(* CODESYS project TerminalApp.project
   Title: Терминал моечного поста
   Version: 0.0.0.1
   Company: ООО АСУ

Project tree, tasks and I/O mapping:
  CompWin : CODESYS Control for Raspberry Pi SL, 3S - Smart Software Solutions GmbH, version 3.5.11.60
    application AppTerminalPost
      libraries: Standard, * (System); Serial Communication, 3.5.7.0 (3S - Smart Software Solutions GmbH); Memory, 3.5.7.0 (3S - Smart Software Solutions GmbH); VisuDialogs, * (System); Time and Date, 3.5.7.0 (3S - Smart Software Solutions GmbH); BASIC, 3.3.3.0 (OSCAT); Standard64, * (System); Util, * (System); SysCom, 3.5.5.0 (System); SysProcess, 3.5.7.0 (System); SysTypes Interfaces, 3.5.2.0 (System); CmpChecksum, 3.5.5.0 (System); SysTime, 3.5.9.0 (System); CmpLog, 3.5.5.0 (System); Component Manager, * (System); CmpErrors Interfaces, * (System); CmpApp, 3.5.13.0 (System); File Access, 3.5.7.0 (3S - Smart Software Solutions GmbH); CmpCharDevice, 3.5.4.0 (3S - Smart Software Solutions GmbH)
      task MainTask (cyclic, interval 100 ms, priority 2) calls PLC_PRG, DeviceButtons, DeviceOut, SafePrg
      task TaskDevBanknote (cyclic, interval 4 ms, priority 1) calls DeviceBanknote [New Cash]
      task TaskDevCoin (cyclic, interval 5 ms, priority 4) calls DeviceCoin
      task TaskDevCard (cyclic, interval t#20ms, priority 3) calls DeviceCard
      task TaskDBG (cyclic, interval t#20ms, priority 1) calls DBG_PRG
      task NVLTask (cyclic, interval t#20ms, priority 1) calls DataToSpk, DataToUI, DataFromSpk
      task TaskPrinter (cyclic, interval t#20ms, priority 31) calls DevicePrinter
      program PLC_PRG [ST]: GetCurrentTime, SetValidComPorts, ControlCodesys
      Symbols
      data type EnumStatePost
      data type AppStatus
      Cash/
        program DeviceBanknote [ST]: GetCounterBanknote, IsCasetteDropped, IsBanknoteJammed, CollectCash, GetReceived
        data type CASHCODE_STATE
        data type CCNET_STATE
        function block COM_CONTROL [ST]: CLOSE, OPEN, SETTINGS
        data type _4BYTES_TO_REAL
        function _BUFFER_CLEAR [ST]
        data type _WORD_TO_2BYTES
        function block ANALYZE_DATA [ST]
        function BYTE_TO_STRH [ST]
        function block CashCode [ST]: CHECK_RESPONSE, GET_DATA_FROM_RESPONSE, GetCRC16, SET_ACK, SET_ENABLE_BILL_TYPES, SET_NSC, SET_PAKET, SET_POLL, SET_RESET, resetMoneyReceived, resetMoneyCnt
        data type COM_STATE
        data type DCON_STATE
        data type SET_4TM_STATE
        data type cacheCodeStatus
        data type CACHECODE_ERROR
        data type devBank
      DevCoin/
        program DeviceCoin [ST]: GetReceived, DbgInCoin, CollectCash, GetCounterCoin
        function block ccTalk [ST]: init, iterateAndUpdateStatus
        data type ccTalkStatus
        data type CCTALK_COIN_TYPES
        data type CCTALK_ERROR
        function block ccTalkSimpleCommand [ST]
        function block ccTalkReadBufferedCreditCommand [ST]
        data type ccTalkEvent
        function ccTalkCRC [ST]
        function ccTalkProcessReadBufferCreditTable [ST]
        function ccTalkGetNoDataCommandBuffer [ST]
      DevCard/
        function block Cards [ST]
        data type EnumCardType
        program DeviceCard [ST]: UnLockCard, DbgSetCard, GetTypeCard, TestValidComPort
        function block crt [ST]: init, iterateAndUpdateStatus, latchLock, latchRelease
        data type crtStatus
        data type CRT_CARD_STATE
        data type CRT_ERROR
        data type crtParametrizedCommand
        function block crtSimpleCommand [ST]
        function crtDecodeCardState [ST]
        function crtBCC [ST]
        function block crtInitCommand [ST]
      global variables GVL
      Debug/
        data type DebugStruct
        program DBG_PRG [ST]: GetInCoin, SetMode, GetInBanknote, UnLockCard
      DevButtons/
        program DeviceButtons [ST]: GetActiveButton
        data type EnumButton
      DevLamps/
        program DeviceLamps [ST]: SetLamps, SetAlarmLamps, SetIllumination, SetLampColor, SetLightTurbo
      Post/
        function block Post [ST]: ChangeMode, AddMoney, RemAmount, ResetModes, FormatModeFinInfo, StartWash, StopWash, SetCard, AvialableCardWork, InWaitModes, IsUnlocked, UnLock, IsReadyToWash, Init, EndCollectCash, BegCollectCash, EndFreemoney, BegFreemoney, InStopMode, OnFinButton, GeFundFromCollect, OnLowPower, SaveRetainVars, RestoreRetainVars, Shutdown, GetMessageInCash, GetMessageFunc, GetMessageCollect, GetFundTotal, GetRates, SaveNewRates, InPaidWashMode, InClearWashMode, GetMessageTotal, InServiceMode, SetSavedFund, SaveNewPause, GetPauseActiveClean, GetPauseFoam, GetPauseShampoo, SetLastInCash
        data type EnumMode
        function block EventMode [ST]: SetValues, ResetValues, StartMode, StopMode
        data type EnumLock
        program SafePrg [ST]
      Config/
        data type EnumInit
        function Initialisation [ST]
        function InitConfiguration [ST]
        function PostParamInit [ST]
        function PostStateInit [ST]
      DevOut/
        global variables NVL2UI
        program DeviceOut [ST]: SetOut
      global variables NVL_TO_SPK
      declarations NVL_FROM_SPK
      Traffic/
        program DataToSpk [ST]
        program DataFromSpk [ST]: GetConfirmedMode, GetAllowedButton, GetBonusValue, GetAllowedMode
        program DataToUI [ST]
      DevPrinter/
        data type PRINTER_FONT_CPI
        data type PRINTER_ERROR
        data type TEXT_ALIGNMENT
        data type PRINTER_FONT
        data type PRINTER_FONT_SIZE
        program DevicePrinter [ST]: printEncashment, PrintBill
        function block printReceipt [ST]
        function unicode2cp866 [ST]
        function unicodeSymbol2cp866 [ST]
        function block receiptBuffer [ST]: setFontCPI, setFontSize, clear, print, push_back, newline, push_back_array, setCP866Encoding, totalCut, initPrinter, ejectTicket, presentPageAndTimeoutRetract, setFontBold, setFontAlignment, println, printWithLeftPadding, print2Colsln, setFont, setFontSize2
      global variables SPK_DATA
      global variables PersistentVars
      program RetainManager [ST]
      function block StdLogger [ST]: AddLogEntry, debug, error, FB_Exit, FB_Init, info, warn
    SoftMotion General Axis Pool
    I²C
      I2C_master : I2C master, 3S - Smart Software Solutions GmbH, version 1.0.0.0
        UBRAIN1 : UBRAIN1, OOO ASU, version 1.1.0.0
            settings: I²C address = 5
    SPI
    GPIOs_A_B : GPIOs A/B, 3S - Smart Software Solutions GmbH, version 3.5.16.0
        unmapped channels: digital inputs (GPIO0..GPIO31), digital outputs (GPIO0..GPIO31)
    Onewire
    Camera device
      <Empty>
    Ethernet : Ethernet, 3S - Smart Software Solutions GmbH, version 3.5.16.0
        settings: IPAddress = [0,0,0,0]; SubnetMask = [0,0,0,0]; GatewayAddress = [0,0,0,0]; MACAddress = [16#00,16#00,16#00,16#00,16#00,16#00]; NetworkInterfaceName = 'eth0'; NetworkInterfaceName = "eth0"; SaveCommunicationSettings = FALSE
      ModbusTCP_Slave_Device : ModbusTCP Slave Device, 3S - Smart Software Solutions GmbH, version 3.5.16.0
          input  AppTerminalPost.SPK_DATA.gi_aAllowedFlags[0] : BOOL  // Регистры временного хранения.Регистры временного хранения.Bit0
          input  AppTerminalPost.SPK_DATA.gi_aAllowedFlags[1] : BOOL  // Регистры временного хранения.Регистры временного хранения.Bit1
          input  AppTerminalPost.SPK_DATA.gi_aAllowedFlags[2] : BOOL  // Регистры временного хранения.Регистры временного хранения.Bit2
          input  AppTerminalPost.SPK_DATA.gi_aAllowedFlags[3] : BOOL  // Регистры временного хранения.Регистры временного хранения.Bit3
          input  AppTerminalPost.SPK_DATA.gi_aAllowedFlags[4] : BOOL  // Регистры временного хранения.Регистры временного хранения.Bit4
          input  AppTerminalPost.SPK_DATA.gi_aAllowedFlags[5] : BOOL  // Регистры временного хранения.Регистры временного хранения.Bit5
          input  AppTerminalPost.SPK_DATA.gi_aAllowedFlags[6] : BOOL  // Регистры временного хранения.Регистры временного хранения.Bit6
          input  AppTerminalPost.SPK_DATA.gi_aAllowedFlags[7] : BOOL  // Регистры временного хранения.Регистры временного хранения.Bit7
          input  AppTerminalPost.SPK_DATA.gi_nCurFunction : WORD  // Регистры временного хранения.Регистры временного хранения
          output AppTerminalPost.SPK_DATA.go_postFunction : WORD  // Входные регистры.Входные регистры
          output AppTerminalPost.SPK_DATA.go_postCounterFund : WORD  // Входные регистры.Входные регистры
          unmapped channels: Регистры временного хранения, Входные регистры
  libraries: VisuSymbols, 3.5.10.0 (System)
  text list GlobalTextList
*)

// CompWin/AppTerminalPost/EnumStatePost
// Состояния поста
{attribute 'qualified_only'}
{attribute 'strict'}
TYPE EnumStatePost :
(
	IDLE	:= 0,	// Экран ожидания
	ADVERT	:= 100,	// Экран показа рекламы
	CARD	:= 200,	// Экран клиентской карты
	CASH	:= 300,	// Экран внесения денежных средств
	FUNC	:= 400,	// Экран функций
	FIN		:= 500,	// Экран окончания мойки
	CLEANUP	:= 600,	// Экран уборки
	ENCASH	:= 700,	// Экран инкассации
	STOP	:= 1000	// Экран состояния останова поста
);
END_TYPE

// CompWin/AppTerminalPost/Post/EnumMode
// Функции мойки
{attribute 'qualified_only'}
{attribute 'strict'}
TYPE EnumMode :
(
	FUNC		:= 0,	// терминал готов к включению функций
	
	ACTIVECLEAN	:= 1,	// Р1. ECO-power		2
	FOAM		:= 2,	// Р2. Пена				4
	SHAMPOO		:= 3,	// Р3. Шампунь			3
	COLDWATER	:= 4,	// Р4. Холодная вода	1
	HOTWATER	:= 5,	// Р5. Горячая вода		2
	WAX			:= 6,	// Р6. Воск				4
	OSMOSE		:= 7,	// Р7. Осмос			3
	PAUSE		:= 8,	// Пауза				4
	HIGHPRESSURE := 14, // ХВ высокого давления 
	
	IDLE		:= 9,	// терминал в ожидании клиентов
	ADVERT		:= 10,	// реклама	
	
	FIN			:= 500,	// Экран окончания мойки
	CLEANUP		:= 600,	// Экран уборки
	CASHCOLLECT	:= 700,	// Экран инкассации
	CASHCOLLECT_FIN	:= 710,	// Экран окончания инкассации
	FREEMONEY	:= 800,	// Экран добавления денег
	STOP		:= 1000	// Экран состояния останова поста

//	CARD	:= 200,	// Экран клиентской карты
//	CASH	:= 300,	// Экран внесения денежных средств
);
END_TYPE

// CompWin/AppTerminalPost/Config/EnumInit
// Кода возврата процедуры инициализации
{attribute 'qualified_only'}
{attribute 'strict'}
TYPE EnumInit :
(
	INIT_RET_FAIL       := 0, //      0 - инициализация закончилась с ошибкой
	INIT_RET_SUCC_RESET := 1, //      1 - инициализация успешно проведена, требуется перезапуск
	INIT_RET_SUCC       := 2, //      2 - инициализация успешно проведена, перезапуск не требуется
	INIT_RET_NO         := 3  //      3 - в инициализации не было необходимости
);
END_TYPE

// CompWin/AppTerminalPost/AppStatus
// Состояние приложения
TYPE AppStatus :
STRUCT
	startFlag: BOOL := TRUE;	// флаг начального запуска
	infoString: STRING := 'Starting ...';	// информация о состоянии приложения
	rebootFlag : BOOL := FALSE;	// флаг необходимости перезапуска
	
	errNimber: INT := 0;
	errString: STRING;
END_STRUCT
END_TYPE

// CompWin/AppTerminalPost/DevCard/EnumCardType
// Типы карт
{attribute 'qualified_only'}
{attribute 'strict'}
TYPE EnumCardType :
(
	UNDEFINED	:= 0,	// неопределённая карта (карта отсутствует)
	CLEANUP		:= 1,	// карта уборки
	CASHCOLLECT	:= 2,	// карта инкассации
	FREEMONEY	:= 3,	// карта добавления денег (бесплатной мойки)
	SERVICE		:= 4	// карта техслужбы
);
END_TYPE

// CompWin/AppTerminalPost/Cash/CASHCODE_STATE

TYPE CASHCODE_STATE :
(
	INIT,
	DISABLE,
	RESET,
	POLL,
	ENABLE_BILL_TYPES
);
END_TYPE

// CompWin/AppTerminalPost/Cash/CCNET_STATE

TYPE CCNET_STATE :
(
	INIT,
	IDLE,
	SEND_POLL,
	SEND_ENABLE_BILL_TYPES,
	SEND_COMMAND, //Command transmission
	SEND_ASC, //Подтверждаем получение
	SEND_NSC, //Не подтверждааем получение
	SEND_RESET, //reset
	RECEIVE_RESPONSE,
	RESPONSE_DELAY,
	WAIT_ENROLLMENT,
	WAIT_WRITE,
	POLLING_CYCLE_ENDS
	
	
);
END_TYPE

// CompWin/AppTerminalPost/DevCoin/ccTalkStatus
///element of ccTalk ReadBufferCredit (229) command output
TYPE ccTalkStatus :
STRUCT
	coinsReceived : ARRAY[0..5] OF BYTE;  //принятые монеты по номиналам
	coinsRejected : UINT;   //непринятые монеты
	moneyReceived : UINT;   //денег принято всего
	busy : BOOL := FALSE;  //cannot execute command
	error: CCTALK_ERROR;

	// количество монет в боксе
	countCoin: UINT := 0;
	// количества монет по номиналам
	receivedCoin1: UINT := 0;
	receivedCoin2: UINT := 0;
	receivedCoin5: UINT := 0;
	receivedCoin10: UINT := 0;
END_STRUCT
END_TYPE

// CompWin/AppTerminalPost/DevCoin/CCTALK_COIN_TYPES
TYPE CCTALK_COIN_TYPES :
(
//	COIN_1RUB := 16#1000 OR 16#0800,
//	COIN_2RUB := 16#4000 OR 16#2000,
//	COIN_5RUB := 16#0001 OR 16#8000,
//	COIN_10RUB := 16#0004 OR 16#0002

//	COIN_1RUB := 16#1000 OR 16#0800,
//	COIN_2RUB := 16#4000 OR 16#2000,
//	COIN_5RUB := 16#0001 OR 16#8000,
//	COIN_10RUB := 16#0001 OR 16#8000
	COIN_10RUB := 16#FFFF
	
) UINT;
END_TYPE

// CompWin/AppTerminalPost/DevCoin/CCTALK_ERROR
{attribute 'strict' := ''}
TYPE CCTALK_ERROR :
(
	CCTALK_NO_ERROR,
	CCTALK_OPEN_ERROR,
	CCTALK_INIT_PROC_NOT_CALLED
) BYTE;
END_TYPE

// CompWin/AppTerminalPost/DevCoin/ccTalkEvent
///element of ccTalk ReadBufferCredit (229) command output
TYPE ccTalkEvent :
STRUCT
	validationChannel: BYTE;
	errorCode: BYTE;
END_STRUCT
END_TYPE

// CompWin/AppTerminalPost/DevCard/crtStatus
///element of ccTalk ReadBufferCredit (229) command output
TYPE crtStatus :
STRUCT
	cardState: CRT_CARD_STATE := CRT_CARD_UNDEFINED;
	///cannot execute command
	busy: BOOL := FALSE;
	///is latch locked ?
	locked: BOOL := FALSE;
	error: CRT_ERROR;
	isInit : BOOL;
END_STRUCT
END_TYPE

// CompWin/AppTerminalPost/DevCard/CRT_CARD_STATE
{attribute 'strict' := ''}
TYPE CRT_CARD_STATE :
(
	CRT_CARD_UNDEFINED,
	CRT_CARD_INSIDE,
	CRT_RF_CARD_INSIDE,
	CRT_NO_CARD
);
END_TYPE

// CompWin/AppTerminalPost/DevCard/CRT_ERROR
{attribute 'strict' := ''}
TYPE CRT_ERROR :
(
	CRT_NO_ERROR,
	CRT_OPEN_ERROR,
	CRT_INIT_PROC_NOT_CALLED
);
END_TYPE

// CompWin/AppTerminalPost/DevCard/crtParametrizedCommand
///command and parameter for using in CRT protocol
TYPE crtParametrizedCommand :
STRUCT
	CM: BYTE;
	PM: BYTE;
END_STRUCT
END_TYPE

// CompWin/AppTerminalPost/Debug/DebugStruct
// Структура отладочной визуализации
TYPE DebugStruct :
STRUCT
//	Mode: EnumMode := EnumMode.WAIT;
	
	InBanknote: WORD := 0;
	
	InCoin: WORD := 0;
	
	CardType: EnumCardType := EnumCardType.UNDEFINED;
END_STRUCT
END_TYPE

// CompWin/AppTerminalPost/Cash/_4BYTES_TO_REAL
TYPE _4BYTES_TO_REAL :
UNION
	rValue :REAL;
	abyModbusReal : ARRAY [0..3] OF BYTE;
END_UNION
END_TYPE

// CompWin/AppTerminalPost/DevButtons/EnumButton
// функциональные кнопки
{attribute 'qualified_only'}
{attribute 'strict'}
TYPE EnumButton :
(
	NONE := 0,				// нет нажатой кнопки
	BTN_SHAMPOO := 1,		// Шампунь
	BTN_ACTIVECLEAN := 2,	// ECO-power
	BTN_FOAM := 3,			// Пена
	BTN_COLDWATER := 4,		// Холодная вода
	BTN_HOTWATER := 5,		// Горячая вода
	BTN_WAX := 6,			// Воск
	BTN_OSMOSE := 7,		// Осмос
	BTN_PAUSE := 8,			// Пауза
	BTN_PRINT := 9,			// Печать чека
	BTN_HIGHPRESSURE := 10	// Вызов оператора
);
END_TYPE

//VAR CONSTANT
//	BTN_FUNC_FIRST :BYTE := 1;
//	BTN_FUNC_LAST :BYTE := 8;
//	BTN_FIRST :BYTE := 1;
//	BTN_LAST :BYTE := 10;
//END_VAR

// CompWin/AppTerminalPost/Post/EnumLock
// замки поста
{attribute 'qualified_only'}
{attribute 'strict'}
TYPE EnumLock :
(
	LOCK_TOP := 1,	// 2#0100_0000,		// верхний замок
	LOCK_MID := 2	// 2#1000_0000		// средний замок
);
END_TYPE

// CompWin/AppTerminalPost/DevPrinter/PRINTER_FONT_CPI
{attribute 'strict' := ''}
TYPE PRINTER_FONT_CPI :
(
	CPI_SMALL := 0,
	CPI_BIG := 1,
	CPI_MEDIUM := 2
) BYTE;
END_TYPE

// CompWin/AppTerminalPost/DevPrinter/PRINTER_ERROR
{attribute 'strict' := ''}
TYPE PRINTER_ERROR :
(
	PRINTER_NO_ERROR,
	PRINTER_FILE_OPEN_ERROR,
	PRINTER_WRITE_ERROR
) BYTE;
END_TYPE

// CompWin/AppTerminalPost/DevPrinter/TEXT_ALIGNMENT
{attribute 'strict' := ''}
TYPE TEXT_ALIGNMENT :
(
	ALIGN_LEFT := 0,
	ALIGN_CENTER := 1,
	ALIGN_RIGHT := 2
) BYTE;
END_TYPE

// CompWin/AppTerminalPost/DevPrinter/PRINTER_FONT
{attribute 'strict' := ''}
TYPE PRINTER_FONT :
(
	FONT_A := 0,
	FONT_B := 1
) BYTE;
END_TYPE

// CompWin/AppTerminalPost/DevPrinter/PRINTER_FONT_SIZE
{attribute 'strict' := ''}
TYPE PRINTER_FONT_SIZE :
(
	FONT_SMALL := 1,
	FONT_BIG := 0
) BYTE;
END_TYPE

// CompWin/AppTerminalPost/Cash/_WORD_TO_2BYTES
TYPE _WORD_TO_2BYTES :
UNION
	wValue : WORD;
	abyWord : ARRAY [0..1] OF BYTE;
END_UNION
END_TYPE

// CompWin/AppTerminalPost/Cash/COM_STATE
TYPE COM_STATE :
(
	INITIALIZE := 00,
	WAITING_FOR_SIGNAL := 10,
	OPEN_PORT := 20,
	CLOSE_PORT := 30
);
END_TYPE

// CompWin/AppTerminalPost/Cash/DCON_STATE

TYPE DCON_STATE :
(
	CREATE_REQUEST := 00,
	SEND_REQUEST := 10,
	RECEIVE_RESPONSE := 20,
	RESPONSE_DELAY := 30,
	POLLING_CYCLE_ENDS := 40
);
END_TYPE

// CompWin/AppTerminalPost/Cash/SET_4TM_STATE
TYPE SET_4TM_STATE :
(
	CREATE_CHANNEL := 00,
	OPEN_CHANNEL := 10,
	RECEIVE_CHANNEL := 20,
	RESPONSE_DELAY_CHANNEL := 30,
	CREATE_REQUEST := 40,
	SEND_REQUEST := 50,
	RECEIVE_RESPONSE := 60,
	RESPONSE_DELAY := 70,
	POLLING_CYCLE_ENDS := 80
);
END_TYPE

// CompWin/AppTerminalPost/Cash/cacheCodeStatus
///element of ccTalk ReadBufferCredit (229) command output
TYPE cacheCodeStatus :
STRUCT
	///принятая купюра
	moneyReceived: UINT;
	///cannot execute command
	busy: BOOL := FALSE;
	error: CACHECODE_ERROR;
//	// количество купюр в боксе
//	countBanknote: UINT := 0;
	// состояние купюрника
	cashcodeStatus : WORD := 0;
	// ошибка купюрника
	cashcodeError : WORD := 0;

	// флаг снятия касетты
	casetteDropped : WORD := 0;
	// флаг зажёвывания банкноты
	banknoteJammed : WORD := 0;
	
	// количества купюр по номиналам
	receivedBanknote10: UINT := 0;
	receivedBanknote50: UINT := 0;
	receivedBanknote100: UINT := 0;
	receivedBanknote500: UINT := 0;
	receivedBanknote1000: UINT := 0;
	receivedBanknote5000: UINT := 0;
END_STRUCT
END_TYPE

// CompWin/AppTerminalPost/Cash/CACHECODE_ERROR
TYPE CACHECODE_ERROR :
(
	CACHECODE_NO_ERROR,
	CACHECODE_OPEN_ERROR
);
END_TYPE

// CompWin/AppTerminalPost/Cash/devBank
TYPE devBank :
(
	INIT := 0,
	CLOSE,
	OPEN,
	PROCESS
);
END_TYPE

// CompWin/AppTerminalPost/DevOut/NVL2UI
{attribute 'qualified_only'}
VAR_GLOBAL
	// номер поста
	postNumber: INT;
	
	// Состояние терминала: ожидание, функции, окончание мойки, уборка, инкассация, пополнение баланса оператором
	postMode: INT;
	// TYPE EnumMode :
	// (
	// 	FUNC		:= 0,	// терминал готов к включению функций
	// 	
	// 	ACTIVECLEAN	:= 1,	// Р1. ECO-power		2
	// 	FOAM		:= 2,	// Р2. Пена				4
	// 	SHAMPOO		:= 3,	// Р3. Шампунь			3
	// 	COLDWATER	:= 4,	// Р4. Холодная вода	1
	// 	HOTWATER	:= 5,	// Р5. Горячая вода		2
	// 	WAX			:= 6,	// Р6. Воск				4
	// 	OSMOSE		:= 7,	// Р7. Осмос			3
	// 	PAUSE		:= 8,	// Пауза				4
	// 	
	// 	IDLE		:= 9,	// терминал в ожидании клиентов
	// 	ADVERT		:= 10,	// реклама	
	// 	
	// 	FIN			:= 500,	// Экран окончания мойки
	// 	CLEANUP		:= 600,	// Экран уборки
	// 	CASHCOLLECT	:= 700,	// Экран инкассации
	// 	CASHCOLLECT_FIN	:= 710,	// Экран окончания инкассации
	// 	FREEMONEY	:= 800	// Экран добавления денег
	// 	STOP		:= 1000	// Экран состояния останова поста
	// );
	// END_TYPE

	// баланс
	postCounterFund: INT;

	// тип карты
	cardType: INT;
	// TYPE EnumCardType :
	// (
	// 	UNDEFINED	:= 0,	// неопределённая карта (карта отсутствует)
	// 	CLEANUP		:= 1,	// карта уборки
	// 	CASHCOLLECT	:= 2,	// карта инкассации
	// 	FREEMONEY	:= 3,	// карта добавления денег (бесплатной мойки)
	// 	SERVICE		:= 4	// карта техслужбы
	// );
	// END_TYPE	

	
	// нажатая кнопка
	buttonActive: INT;
	// TYPE EnumButton :
	// (
	// 	NONE := 0,				// нет нажатой кнопки
	// 	BTN_ACTIVECLEAN := 1,	// Р1. ECO-power
	// 	BTN_FOAM := 2,			// Р2. Пена
	// 	BTN_SHAMPOO := 3,		// Р3. Шампунь
	// 	BTN_COLDWATER := 4,		// Р4. Холодная вода
	// 	BTN_HOTWATER := 5,		// Р5. Горячая вода
	// 	BTN_WAX := 6,			// Р6. Воск
	// 	BTN_OSMOSE := 7,		// Р7. Осмос
	// 	BTN_PAUSE := 8,			// Пауза
	// 	BTN_PRINT := 9,			// Печать чека
	// 	BTN_HELP := 10			// Вызов оператора
	// );
	// END_TYPE
		
	// сумма внесения
	amountReceived: INT;
	
	
	// стоимость оконченной мойки
	costWash: INT;
	// сдача
	costChange: INT;
	// стоимость активной химии
	costActiveClean: INT;
	// стоимость пены
	costFoam: INT;
	// стоимость шампуня
	costShampoo: INT;
	// стоимость ХВ
	costColdWater: INT;
	// стоимость ГВ
	costHotWater: INT;
	// стоимость воска
	costWax: INT;
	// стоимость осмоса
	costOsmose: INT;
	// стоимость паузы
	costPause: INT;

	
	// состояние верхнего замка
	lockTop: INT;
	// состояние среднего замка
	lockMid: INT;
	// 1 - замок закрыт; 0 - замок открыт
END_VAR

// CompWin/AppTerminalPost/GVL
{attribute 'qualified_only'}
VAR_GLOBAL
	btn_1: BOOL;
	//cnt_1: INT;
	SetAlarmLamps: INT;
	
	printEncashmentReceipt : BOOL :=FALSE;
	
	glFlagStartVideo : ARRAY[0..10] OF BOOL;
	glFlagStartIdleVideo : BOOL;
	
END_VAR

// CompWin/AppTerminalPost/NVL_TO_SPK
{attribute 'qualified_only'}
VAR_GLOBAL
	// номер поста
	go_postNumber: INT;
	// выбранная функция
	go_postFunction: INT;
	// баланс поста
	go_postCounterFund: INT;
END_VAR

// CompWin/AppTerminalPost/NVL_FROM_SPK
//This gobal variable list is received via the network.
//Sender: Imported from file 'D:\lexadev\ЭкоМойки\gitrep\dev\TerminalController\NVL_Sender.gvl'
//Protocol: UDP

VAR_GLOBAL
	n_iCounter: INT;	
	n_aPostMode: ARRAY [0..5] OF INT;
	n_aAllowedFlags: ARRAY [0..5,1..7] OF BOOL;
END_VAR

// CompWin/AppTerminalPost/SPK_DATA
{attribute 'qualified_only'}
VAR_GLOBAL
	// to SPK
	go_postNumber: INT;
	go_postFunction: INT;
	go_postCounterFund: INT;
	go_counter: UINT;
	
	// from SPK
	gi_nCurFunction: INT;
	gi_aAllowedFlags: ARRAY [0..7] OF BOOL;

	// from AG
	// флаг необходимости применения тарифов от сервера
	// 1 - надо применить тарифы сервера, 0 - игнорировать
	gi_rateSave : WORD;
	
	// новые тарифы режимов от сервера 
	gi_rates : ARRAY [0 .. 8] OF WORD;
	
	// бонусы
	// текущий процент бонусов
	gi_bonusValue: WORD := 0;
	// час начала действия бонусов 24H
	gi_bonusStart: WORD := 22;
	// час окончания действия бонусов 24H
	gi_bonusStop: WORD := 6;
	
	
	// флаг необходимости применения пауз от сервера
	// 1 - надо применить паузы сервера, 0 - игнорировать
	gi_pauseSave : WORD;

	// паузы режимов в секундах
	gi_pauseActiveClean: WORD;
	gi_pauseFoam: WORD;
	gi_pauseShampoo: WORD;
	
	
	// to server
	counterBanknote10: WORD;
	counterBanknote50: WORD;
	counterBanknote100: WORD;
	counterBanknote500: WORD;
	counterBanknote1000: WORD;
	counterBanknote5000: WORD;

	counterCoin: WORD;
	counterCoin1: WORD;
	counterCoin2: WORD;
	counterCoin5: WORD;
	counterCoin10: WORD;
	
	// внесений с инкассации
	fundFromCollect: UINT;
	// внесений с начала работы
	fundTotal: UINT;

//	messageInCash: STRING;
//	messageFunc: STRING;
//	messageCollect: STRING;
	messageInCash: ARRAY[0..64] OF WORD;
	messageFunc:  ARRAY[0..64] OF WORD;
	messageCollect:  ARRAY[0..64] OF WORD;
	messageTotal:  ARRAY[0..64] OF WORD;
	
	// текущие тарифы
	currentRates : ARRAY[0..8] OF WORD;

	// ФЛАГИ КУПЮРНИКА
	// состояние купюрника
	cashcodeStatus : WORD := 0;
	// ошибка купюрника
	cashcodeError : WORD := 0;
	
	// флаг инкассации (отсоединения касетты)
	casetteDropped : WORD := 0;
	// флаг зажёвывания банкноты
	banknoteJammed : WORD := 0;
	
	// Флаги блокировки дверей
	lockTop : WORD := 1;
	lockMid : WORD := 1;
	
	// паузы режимов в секундах
	currentPauseActiveClean: WORD;
	currentPauseFoam: WORD;
	currentPauseShampoo: WORD;
END_VAR

// CompWin/AppTerminalPost/PersistentVars
{attribute 'qualified_only'}
VAR_GLOBAL PERSISTENT RETAIN
	// тотальная несбрасываемый счётчик выручки
	TotalFund : UINT := 0;	
	
	// total количества купюр по номиналам
	totalBanknote10: DWORD := 0;
	totalBanknote50: DWORD := 0;
	totalBanknote100: DWORD := 0;
	totalBanknote500: DWORD := 0;
	totalBanknote1k: DWORD := 0;
//	totalBanknote5000: DWORD := 0;

	// total количества монет по номиналам
//	totalCoin1: DWORD := 0;
//	totalCoin2: DWORD := 0;
//	totalCoin5: DWORD := 0;
	totalCoin10: DWORD := 0;

	//// выручка в посту (сбрасывается при инкассации)
	//CashFund : UINT := 0;
	
	// количества купюр по номиналам
	counterBanknote10: UINT := 0;
	counterBanknote50: UINT := 0;
	counterBanknote100: UINT := 0;
	counterBanknote500: UINT := 0;
	counterBanknote1000: UINT := 0;
//	counterBanknote5000: UINT := 0;

	// количества монет по номиналам
//	counterCoin1: UINT := 0;
//	counterCoin2: UINT := 0;
//	counterCoin5: UINT := 0;
	counterCoin10: UINT := 0;
	
	// количества купюр по номиналам до инкассации
	counterBefCollectBanknote10: UINT := 0;
	counterBefCollectBanknote50: UINT := 0;
	counterBefCollectBanknote100: UINT := 0;
	counterBefCollectBanknote500: UINT := 0;
	counterBefCollectBanknote1000: UINT := 0;
//	counterBefCollectBanknote5000: UINT := 0;

	// количества монет по номиналам до инкассации
//	counterBefCollectCoin1: UINT := 0;
//	counterBefCollectCoin2: UINT := 0;
//	counterBefCollectCoin5: UINT := 0;
	counterBefCollectCoin10: UINT := 0;
//	messageCollectCoin : STRING := '';
	
	// сообщение о внесении
	messageInCash: STRING[130] := '';
	// сообщение о функции
	messageFunc: STRING[130] := '';
	// сообщение об инкассации
	messageCollect: STRING[130] := '';
	// сообщение о тотальном счётчике
	messageTotal: STRING[130] := '';
	
	// тарифы функций 
	rates : ARRAY [0 .. 8] OF WORD := [
	2700, 	// ACTIVECLEAN	:= 1,	// Р1. ECO-power
	3300, 	// FOAM		:= ,	// Р2. Пена
	2300, 	// SHAMPOO		:= ,	// Р3. Вода + шампунь
	1500, 	// COLDWATER	:= 4,	// Р4. Холодная вода
	2400, 	// HOTWATER	:= 5,	// Р5. Горячая вода
	3600, 	// WAX			:= 6,	// Р6. Воск
	2700, 	// OSMOSE		:= 7,	// Р7. Осмос
	100,	// PAUSE		:= 8,	// пауза
	2100	// HIGHPRESSURE	:= 9,	// ХВ высокого давления
	];
	
	// сохранённый баланс  с меткой времени
	fundTime : DATE_AND_TIME;
	fundSaved100 : WORD;
	
	// адрес мойки
	washAddress : WSTRING := "Волгоград Жукова 55";
	// номер поста
	postNumber : INT := 0;
	
	// паузы режимов в секундах
	pauseActiveClean: TIME := T#10S;
	pauseFoam: TIME := T#0S;
	pauseShampoo: TIME := T#5S;
	flUseIdleVideo : BOOL := FALSE;
	
END_VAR

// CompWin/AppTerminalPost/PLC_PRG
PROGRAM PLC_PRG
VAR
	appStatus: AppStatus;	// состояние приложения
	
	post: Post;

	timStandbyTime: TIME := T#5S;	//Время в режиме ожидания (c)
	timAdvertisingTime: TIME := T#5S;	//Время в режиме рекламы (c)
	timFinTime: TIME := T#20S;	//Время в экране окончания мойки (c)
	
	timIdleFilterCash:		TIME;	//Фильтр задержки реакции на изменение сигналов внесения и уборки (с)
	timIdleFilterMode:		TIME;	//Фильтр задержки реакции на изменение сигналов режимов (с)
	
	receivedBanknote: WORD;
	receivedCoin: WORD;
	
   	getDT : DTU.GetDateAndTime;
	prevTime : DT;
	currentTime : DT;
	workSecond : DWORD;

	durationSecond: TIME;
	waitSecond: TIME;
	
	//amount : WORD;
	
	comPortCard : BYTE := 0;
	comPortCascode : BYTE := 0;
	
	ii : byte;
	InStopMode: INT;
	
	startTime : DT;
	
	// время начала режимов с задержкой
	startTm_ActiveClean: DT;
	startTm_Foam: DT;
	startTm_Shampoo: DT;
	fDelay: BOOL := FALSE;
	
	//Вспомогательные переменные
	udiResult: UDINT;
	udiTimeLocal : UDINT;
	timeDate: DATE_AND_TIME;
	
	bb : EnumButton;
	
	logger : StdLogger;
END_VAR

// в начале определить текущее время
currentTime := GetCurrentTime();
IF(currentTime > DT#1970-01-01-00:00:00)THEN
	// Начальная инициализация
	IF(appStatus.startFlag) THEN
		appStatus.infoString := Initialisation();
		
		RetainManager(ForceRestore := TRUE, ForceSave := FALSE);
	
		// Включить отладку
		//DBG_PRG.dbgProcess := TRUE;
		DBG_PRG.dbgProcess := FALSE;
		
		// инициализировать пост
		post.Init();
		
		// установить com порты
		SetValidComPorts();
		
		// восстановить сохранённый до перезапуска баланс
//		WHILE((currentTime = DT#1970-01-01-00:00:00) OR (idt < 1000))DO
//			currentTime := GetCurrentTime();
//			idt := idt + 1;
//		END_WHILE
		post.SetSavedFund(PersistentVars.fundTime, PersistentVars.fundSaved100 / 100.0);
	
		appStatus.startFlag := FALSE;
	END_IF
	
	//GVL.cnt_1 := GVL.cnt_1 + 1;
	
	currentTime := GetCurrentTime();
	IF(prevTime = DT#1970-01-01-00:00:00)THEN
		prevTime := currentTime;
	END_IF
	
	IF(startTime = DT#1970-01-01-00:00:00)THEN
		startTime := currentTime;
	END_IF
	
	// действия с периодичностью 1 секунда
	workSecond := TIME_TO_DWORD(currentTime - prevTime) / 1000;
	IF(workSecond > 0)THEN
		prevTime := currentTime;
		
		
	//	FOR ii := 1 TO 8 DO
	//		UBRAIN1.bColorButton[ii - 1] := DeviceLamps.COLOR_GREEN;
	//	END_FOR
	
	// учитывать задержку для определенных режимов	
	IF(NOT fDelay)THEN
		post.RemAmount(workSecond);
	END_IF
	
		// получить принятые купюры
		receivedBanknote := DeviceBanknote.GetReceived(); //xxx
		// получить принятые монеты
		receivedCoin := DeviceCoin.GetReceived();
	
		// увеличить сумму в посте
		//IF(receivedBanknote > 0 OR receivedCoin > 0)THEN
			post.AddMoney(receivedBanknote, receivedCoin);
		//END_IF
		
	//	IF(post.Mode <> DeviceButtons.Mode AND post.CounterFund > 0)THEN
	//		post.ChangeMode(DeviceButtons.Mode);
	//	END_IF
	
		// работа в режиме ожидания
		CASE post.Mode OF
	//		EnumMode.IDLE:
	//			waitSecond := timStandbyTime;
	//			durationSecond := currentTime - post.ModeStartTime;
	//			IF(durationSecond > waitSecond)THEN
	//				post.ChangeMode(EnumMode.ADVERT);
	//			END_IF;
	//		EnumMode.ADVERT:
	//			waitSecond := timAdvertisingTime;
	//			durationSecond := currentTime - post.ModeStartTime;
	//			IF(durationSecond > waitSecond)THEN
	//				post.ChangeMode(EnumMode.IDLE);
	//			END_IF;
			EnumMode.FIN:
				waitSecond := timFinTime;
				durationSecond := currentTime - post.ModeStartTime;
				IF(durationSecond > T#20S)THEN
					post.ChangeMode(EnumMode.IDLE);
				END_IF;
			EnumMode.CASHCOLLECT_FIN:
				waitSecond := timFinTime;
				durationSecond := currentTime - post.ModeStartTime;
				IF(durationSecond > T#5S)THEN
					post.ChangeMode(EnumMode.IDLE);
				END_IF;
		END_CASE
	END_IF
	
	// проверять CODESYS
	IF(post.InWaitModes())THEN
		ControlCodesys();
	END_IF
	
	// пост в останове
	IF(post.InStopMode())THEN
		// подсветка терминала
		DeviceLamps.SetIllumination(DeviceLamps.ILLUMINATION_COLOR_RED);
	END_IF
		
	// из режима ожидания переход к мойке
	IF(post.InWaitModes())THEN
		// подсветка терминала
		DeviceLamps.SetIllumination(DeviceLamps.ILLUMINATION_COLOR_LIGHTBLUE);
		GVL.glFlagStartIdleVideo := TRUE;	
		IF(post.IsReadyToWash()) THEN
			post.ChangeMode(EnumMode.FUNC);
		END_IF
	END_IF
	
	// работа в режиме мойки
	IF(post.IsReadyToWash())THEN
		// подсветка терминала
		IF(post.InClearWashMode())THEN
			// в режиме уборки - жёлтый
			DeviceLamps.SetIllumination(DeviceLamps.ILLUMINATION_COLOR_YELLOW);
		ELSE
			// основная подсветка в режиме мойки - зелёный
			DeviceLamps.SetIllumination(DeviceLamps.ILLUMINATION_COLOR_GREEN);
		END_IF
	
	//	CASE DeviceButtons.GetActiveButton() OF
		CASE DataFromSpk.GetConfirmedMode() OF
			EnumMode.ACTIVECLEAN:
				IF(startTm_ActiveClean = DT#1970-01-01-00:00:00)THEN
					startTm_ActiveClean := currentTime;
					fDelay := TRUE;
				ELSE
					durationSecond := currentTime - startTm_ActiveClean;
					IF(durationSecond >= post.GetPauseActiveClean())THEN
						fDelay := FALSE;
					END_IF;
				END_IF
				post.ChangeMode(EnumMode.ACTIVECLEAN);
			EnumMode.FOAM:
				IF(startTm_Foam = DT#1970-01-01-00:00:00)THEN
					startTm_Foam := currentTime;
					fDelay := TRUE;
				ELSE
					durationSecond := currentTime - startTm_Foam;
					IF(durationSecond >= post.GetPauseFoam())THEN
						fDelay := FALSE;
					END_IF;
				END_IF
				post.ChangeMode(EnumMode.FOAM);
			EnumMode.SHAMPOO:
				IF(startTm_Shampoo = DT#1970-01-01-00:00:00)THEN
					startTm_Shampoo := currentTime;
					fDelay := TRUE;
				ELSE
					durationSecond := currentTime - startTm_Shampoo;
					IF(durationSecond >= post.GetPauseShampoo())THEN
						fDelay := FALSE;
					END_IF;
				END_IF
				post.ChangeMode(EnumMode.SHAMPOO);
			EnumMode.COLDWATER:
				post.ChangeMode(EnumMode.COLDWATER);
			EnumMode.HOTWATER:
				post.ChangeMode(EnumMode.HOTWATER);
			EnumMode.WAX:
				post.ChangeMode(EnumMode.WAX);
			EnumMode.OSMOSE:
				post.ChangeMode(EnumMode.OSMOSE);
			EnumMode.PAUSE:
				post.ChangeMode(EnumMode.PAUSE);
			EnumMode.HIGHPRESSURE:
				post.ChangeMode(EnumMode.HIGHPRESSURE);
	//			IF(PLC_PRG.post.Mode = EnumMode.PAUSE)THEN
	//				post.ChangeMode(EnumMode.FIN);
	//			ELSE
	//				post.ChangeMode(EnumMode.PAUSE);
	//			END_IF
			10:
				// ошибка для выбранного режима
				DeviceLamps.SetAlarmLamps(DeviceButtons.GetActiveButton());
			11:
				// пост в останове
				DeviceLamps.SetAlarmLamps(0);
		END_CASE
		
		// сбросить время начала режимов с задержкой
		IF((DataFromSpk.GetConfirmedMode() <> EnumMode.ACTIVECLEAN) AND (DataFromSpk.GetConfirmedMode() <> EnumMode.FOAM) AND (DataFromSpk.GetConfirmedMode() <> EnumMode.SHAMPOO))THEN
			fDelay := FALSE;
		END_IF
		
		IF((startTm_ActiveClean <> DT#1970-01-01-00:00:00) AND (DataFromSpk.GetConfirmedMode() <> EnumMode.ACTIVECLEAN))THEN
			startTm_ActiveClean := DT#1970-01-01-00:00:00;
		END_IF

		IF((startTm_Foam <> DT#1970-01-01-00:00:00) AND (DataFromSpk.GetConfirmedMode() <> EnumMode.FOAM))THEN
			startTm_Foam := DT#1970-01-01-00:00:00;
		END_IF

		IF((startTm_Shampoo <> DT#1970-01-01-00:00:00) AND (DataFromSpk.GetConfirmedMode() <> EnumMode.SHAMPOO))THEN
			startTm_Shampoo := DT#1970-01-01-00:00:00;
		END_IF
	END_IF
	
	// сбросить время начала режимов с задержкой
	IF(NOT post.IsReadyToWash())THEN
		fDelay := FALSE;
		
		IF(startTm_ActiveClean <> DT#1970-01-01-00:00:00) THEN
			startTm_ActiveClean := DT#1970-01-01-00:00:00;
		END_IF

		IF(startTm_Foam <> DT#1970-01-01-00:00:00) THEN
			startTm_Foam := DT#1970-01-01-00:00:00;
		END_IF

		IF(startTm_Shampoo <> DT#1970-01-01-00:00:00) THEN
			startTm_Shampoo := DT#1970-01-01-00:00:00;
		END_IF
	END_IF
	
	// работа в режиме инкассации
	IF(post.Mode = EnumMode.CASHCOLLECT)THEN
		// из-за путаницы в кнопках в инкассации смотртеь на реально нажатую кнопку DeviceButtons.externalActiveButton 
		bb := DeviceButtons.externalActiveButton;
//		CASE DeviceButtons.GetActiveButton() OF
		CASE bb OF
			1:	//EnumButton.BTN_SHAMPOO:
				//// если пост закрыт, то открыть соответствующий замок
				//IF(NOT post.IsUnlocked(EnumLock.LOCK_TOP))THEN
					post.UnLock(EnumLock.LOCK_TOP, TRUE);
				//END_IF
			3:	//EnumButton.BTN_FOAM:
				//// если пост закрыт, то открыть соответствующий замок
				//IF(NOT post.IsUnlocked(EnumLock.LOCK_MID))THEN
					post.UnLock(EnumLock.LOCK_MID, TRUE);
				//END_IF
			2:	//EnumButton.BTN_ACTIVECLEAN:
				// инкассировать пост
				SysTimeRtcConvertUtcToLocal(SysTimeRtcGet(udiResult), udiTimeLocal);
				timeDate:= UDINT_TO_DT(udiTimeLocal);
		//sssxxx		//DevicePrinter.printEncashment(printingTime := OSCAT_BASIC.UTC_TO_LTIME(timeDate, DST_ENABLE :=0, TIME_ZONE_OFFSET:=DevicePrinter.TIME_ZONE_MINUTES_OFFSET), countBanknote10 := DeviceBanknote.GetCounterBanknote(10), countBanknote50 := DeviceBanknote.GetCounterBanknote(50), countBanknote100 := DeviceBanknote.GetCounterBanknote(100),  countCoin10 := DeviceCoin.GetCounterCoin(0));

				DeviceBanknote.CollectCash(); //xxx
				DeviceCoin.CollectCash();
		END_CASE
	END_IF
	
	// работа в режиме добавления денег (бесплатной мойки)
	IF(post.Mode = EnumMode.FREEMONEY)THEN
		CASE DeviceButtons.GetActiveButton() OF
			EnumButton.BTN_ACTIVECLEAN:
				// добавить 5 рублей
				post.AddMoney(5, 0);
			EnumButton.BTN_FOAM:
				// добавить 10 рублей
				post.AddMoney(10, 0);
			EnumButton.BTN_SHAMPOO:
				// добавить 50 рублей
				post.AddMoney(50, 0);
			EnumButton.BTN_COLDWATER:
				// добавить 100 рублей
				post.AddMoney(100, 0);
	//		EnumButton.BTN_PAUSE:
	//			post.EndFreemoney();
		END_CASE
	END_IF
END_IF

METHOD PUBLIC GetCurrentTime : DATE_AND_TIME
VAR
END_VAR
getDT.xExecute := NOT getDT.xDone;
getDT();
IF getDT.xError THEN
    ; // error handling
END_IF
IF getDT.xDone THEN
    // done without error
	currentTime := getDT.dtDateAndTime;
	 //eTZ := getdt.eTimezone;
END_IF

GetCurrentTime := currentTime;
END_METHOD

METHOD SetValidComPorts : BOOL
VAR_INPUT
END_VAR
VAR
	comPort : BYTE;
	portCard : BYTE := 0;
	portBanknote : BYTE := 0;
END_VAR

//DeviceBanknote.TestValidComPort(1);
//DeviceBanknote.TestValidComPort(2);
//DeviceBanknote.TestValidComPort(3);


//DeviceCard.TestValidComPort(10);
//DeviceCard.TestValidComPort(1);
//DeviceCard.TestValidComPort(2);
//DeviceCard.TestValidComPort(3);

//RETURN;

comPortCard := 2;
comPortCascode := 4;
RETURN;

(*
FOR comPort := 1 TO 10 DO
	IF(portCard = 0 AND comPort <> portBanknote)THEN
		IF(DeviceCard.TestValidComPort(comPort))THEN
			portCard := comPort;
		END_IF
	END_IF
	
	IF(portBanknote = 0 AND comPort <> portCard)THEN
		IF(DeviceBanknote.TestValidComPort(comPort))THEN
			portBanknote := comPort;
		END_IF
	END_IF
END_FOR

IF(portCard <> 0)THEN
	comPortCard := portCard;
END_IF

IF(portBanknote <> 0)THEN
	comPortCascode := portBanknote;
END_IF
*)
END_METHOD

METHOD ControlCodesys : BOOL
VAR

	ct : DATE_AND_TIME;

//    command:STRING:= 'sudo /etc/init.d/codesyscontrol restart; read -n1 -t1;';
//    command:STRING[256]:= 'sudo /etc/init.d/codesyscontrol stop && sudo /etc/init.d/codesyscontrol start && date';
    command:STRING[256]:= 'sudo /etc/init.d/codesyscontrol stop';
//    command:STRING:= 'touch /home/pi/mytest123.txt';
    res: SysCom.RTS_IEC_RESULT;
    outbuf:STRING(1000) := '';

END_VAR

ct := GetCurrentTime();
IF((ct - startTime) > T#60M AND NOT appStatus.rebootFlag) THEN
	appStatus.rebootFlag := TRUE;
	PersistentVars.fundSaved100 := 0;
	PersistentVars.fundTime := ct;
	// сохранить retain в файл
	post.SaveRetainVars();
	// выставить флаг необходимости считывания retain переменных из файла
	RetainManager.ForceRestore := TRUE;
	RetainManager.ForceSave := FALSE;
	appStatus.startFlag := TRUE;
	
//	SysProcess.SysProcessExecuteCommand(command, ADR(res));
	SysProcess.SysProcessExecuteCommand2(pszCommand:=command, pszStdOut:= outbuf, udiStdOutLen:= SIZEOF(outbuf), pResult:= ADR(res)); 
END_IF
END_METHOD

END_PROGRAM

// CompWin/AppTerminalPost/Config/Initialisation
// Основная функция инициализации приложения
FUNCTION Initialisation : STRING
VAR_INPUT
END_VAR
VAR
END_VAR

//// Главные установки
//InitBase();

// Инициализировать параметры и начальные значения поста
IF(InitConfiguration() < EnumInit.INIT_RET_SUCC) THEN
//    SDisplaySetError(0);
	Initialisation := 'Err InitConfiguration()';
    return;
END_IF

// Определить параметры поста
IF(PostParamInit() = 0)THEN
	Initialisation := 'Err PostParamInit()';
    RETURN;
END_IF;


//// Инициализировать прерывания таймера
//InitIRQTimer();
  
//// Инициализировать часы
//TimeInit();
  
// Определить состояние поста
PostStateInit();

Initialisation := 'Started';

END_FUNCTION

// CompWin/AppTerminalPost/Config/InitConfiguration
// Процедура инициализации устройства
FUNCTION InitConfiguration : EnumInit
VAR_INPUT
END_VAR
VAR
END_VAR

(*  // Проверить соответствие размеров буферов и структур
  if(SIZE_BUF_VER != sizeof(version_t))
    return INIT_RET_FAIL;
  
  if(SIZE_BUF_PARAM != sizeof(PostParam_t))
    return INIT_RET_FAIL;
  
  if(SIZE_BUF_STATE != sizeof(PostState_t))
    return INIT_RET_FAIL;

  if(SIZE_BUF_EVENT != sizeof(event_t))
    return INIT_RET_FAIL;
  

  // Проверить необходимость инициализации
  if(EEPROM_INIT_CODE == 0x00)
    return INIT_RET_NO;
  
  // Прописать версию ПО
  if(EEPROM_INIT_CODE & INIT_VER)
  {
    if(!MemIntWriteVersion(VERSION))
      return INIT_RET_FAIL;
  }
  
  // Прописать параметры поста
  if(EEPROM_INIT_CODE & INIT_PARAM)
  {
    if(!MemIntWritePostParam(pp))
      return INIT_RET_FAIL;
  }
  
  // Сбросить сохранённое состояние
  if(EEPROM_INIT_CODE & INIT_STATE)
  {
    if(!MemIntWritePostState(ps))
      return INIT_RET_FAIL;
  }
  
  // Сбросить кольцевой буфер, прописав ID следующего события и счётчики
  if(EEPROM_INIT_CODE & INIT_RB)
  {
    // если будет использована флэшка, то очищать её
    #ifdef MEM_FLASH
      MemFlashErase();
    #endif  // MEM_FLASH
      
    // Прописать инициализирующее событие
    uint32_t address = 0;
    #ifdef MEM_INT
      address = FADDR_INT_startRingBuffer;
    //#elif defined MEM_FLASH
    //  address = 0;
    #endif
    MemWriteEvent(address, e, 0);
    
    // Установить количество событий, сохранённых в кольцевом буфере, в 1
    MemIntWriteCountEvents(1);
  }
  
  // Сбросить состояние необходимости инициализации
  EEPROM_INIT_CODE = 0x00;
*)  
  InitConfiguration := EnumInit.INIT_RET_SUCC;

END_FUNCTION

// CompWin/AppTerminalPost/Config/PostParamInit
// Прочитать параметры поста
FUNCTION PostParamInit : BYTE
VAR_INPUT
END_VAR
VAR
END_VAR

  (*uint8_t pbuf[SIZE_BUF_PARAM];

  uint16_t address = FADDR_PARAM;
  
  for(int i = 0; i < sizeof(PostParam_t); i++)
  {
    pbuf[i] = FLASH_ReadByte(address + i);
  }
 
  memcpy(pparam, pbuf, sizeof(PostParam_t));
*)

PostParamInit := 1;

END_FUNCTION

// CompWin/AppTerminalPost/Config/PostStateInit
// Определить состояние поста
FUNCTION PostStateInit : BYTE
VAR_INPUT
END_VAR
VAR
END_VAR

(*
//  PostStateReset();
  
  PostStateRead();
  
  // При запуске всегда нет текущего режима (на флэшке сохранены только закончившиеся режимы)
  // Если не состояние уборки, то считаем, что платный режим
  PMResetCurrentMode(postState.stateKind != 2);
  
  event_t evnt;
  if(RBInitLastEventWithCounters(&evnt))
  {
    // Определить последнее внесение денег
    postState.counterBanknote = evnt.attrCash.counterBanknote;
    postState.counterCoin = evnt.attrCash.counterCoin;
  }

  switch(postState.stateKind)
  {
    case 1:
      // Продолжить сохранённое оставшееся оплаченое время
      if(postState.timerRemain > 0)
        PostTimerIncrement(postState.timerRemain);
      break;
    case 2:
      PMModeFreeSet(1);
      break;
    case 3:
      SDisplaySetCounter(postState.counterBanknote);
      break;
    case 4:
      SDisplaySetCounter(postState.counterCoin);
      break;
  }
*)

PostStateInit := 1;

END_FUNCTION

// CompWin/AppTerminalPost/RetainManager
PROGRAM RetainManager

VAR_INPUT
   RetainFilePathName : STRING := '/home/pi/ASU/AppTerminalPost.ret';
   SaveFilterTime : TIME := T#300MS;
   ForceSave : BOOL;
   ForceRestore : BOOL := TRUE;
   ForceBalance : BOOL := FALSE;
END_VAR
VAR
   pRetainFilePathName : POINTER TO STRING;
   pCurrentApp : POINTER TO APPLICATION;
   RetainAreaSize: __XWORD;
   pRetainArea: POINTER TO BYTE;
   dwCRCSave: DWORD;
   dwCRC: DWORD;
   TOF1 : TOF := (PT := SaveFilterTime);
   R_TRIG1: R_TRIG;
   AppGetCurrent: INT;
   
   
	synccmd: STRING := 'sync -f /home/pi/ASU/AppTerminalPost.ret';
	msg: WSTRING(255);
END_VAR
VAR_OUTPUT
   RTSIECResult : RTS_IEC_RESULT;   
   AttemptSaveCounter: INT;
   Init: BOOL := FALSE;
END_VAR

IF ForceRestore THEN
   pCurrentApp := CmpApp.AppGetCurrent(ADR(RTSIECResult));
   IF RTSIECResult<>0 THEN RETURN; END_IF
   RetainAreaSize := AppGetAreaSize(pApp:= pCurrentApp, uiType:= DA_RETAIN, pResult:= ADR(RTSIECResult));
   IF RTSIECResult<>0 THEN RETURN; END_IF
   pRetainArea := AppGetAreaAddress(pApp:= pCurrentApp, uiType:= DA_RETAIN, pResult:= ADR(RTSIECResult));
   IF RTSIECResult<>0 THEN RETURN; END_IF
   IF LEN(RetainFilePathName) <> 0 THEN
      pRetainFilePathName := ADR(RetainFilePathName);
   ELSE
      pRetainFilePathName := ADR(pCurrentApp^.szName);   
   END_IF
   RTSIECResult := AppRestoreRetainsFromFile(pCurrentApp, pRetainFilePathName^);   
	msg := "ForceRestore";
	PLC_PRG.logger.debug(msg);
   CASE RTSIECResult OF
      0: // #define ERR_OK 0x0000
			msg := "ForceRestore: ERR_OK";
			PLC_PRG.logger.debug(msg);
      16#1E: // #define ERR_SIGNATURE_MISMATCH 0x001E   /* Signature mismatch of an api function */
			msg := "ForceRestore: Signature mismatch of an api function";
			PLC_PRG.logger.debug(msg);
      16#32: // #define ERR_FILE_ERROR 0x0032   /* File error. e.g. cannot open a file for writing because it could be write protected */
			msg := "ForceRestore: File error. e.g. cannot open a file for writing because it could be write protected";
			PLC_PRG.logger.debug(msg);
   ELSE RETURN;
   END_CASE
   dwCRCSave := CRC32Finish(ulCRC:= CRC32Update(ulCRC:= CRC32Init(), pData:= pRetainArea, ulSize:= RetainAreaSize));
   //ForceRestore := FALSE;   
   Init := TRUE;
END_IF

// Запомнить текущий баланс
//IF(PersistentVars.fundSaved100 <> 0 OR REAL_TO_WORD(100 * PLC_PRG.post.CounterFund) <> 0)THEN
(*
IF(Init AND ForceSave)THEN
	IF(PLC_PRG.post.CounterFund > 0)THEN
		PersistentVars.fundSaved100 := REAL_TO_WORD(100 * PLC_PRG.post.CounterFund);
		PersistentVars.fundTime := PLC_PRG.post.ModeStartTime;
//		PersistentVars.fundTime := PLC_PRG.GetCurrentTime();
	ELSE
		PersistentVars.fundSaved100 := 0;
		PersistentVars.fundTime := DT#1970-01-01-00:00:00;
	END_IF
END_IF
*)
IF(Init AND ForceSave AND ForceBalance)THEN
		PersistentVars.fundSaved100 := REAL_TO_WORD(100 * PLC_PRG.post.CounterFund);
		PersistentVars.fundTime := PLC_PRG.GetCurrentTime();
END_IF

R_TRIG1(CLK :=(Init AND ForceSave));
(*
	// количества купюр по номиналам
	PersistentVars.counterBanknote10 := 0;
	PersistentVars.counterBanknote50 := 67;
	PersistentVars.counterBanknote100 := 75;
	PersistentVars.counterBanknote500 := 0;
	PersistentVars.counterBanknote1000 := 0;

	PersistentVars.counterCoin10 := 173;
	
	
	// total количества купюр по номиналам
	PersistentVars.totalBanknote10 := 54;
	PersistentVars.totalBanknote50 := 579;
	PersistentVars.totalBanknote100 := 618;
	PersistentVars.totalBanknote500 := 0;
	PersistentVars.totalBanknote1k := 1;

	// total количества монет по номиналам
	PersistentVars.totalCoin10 := 181;

PersistentVars.TotalFund := PLC_PRG.post.GeFundFromCollect(); 

PersistentVars.rates[0] := 2700;
PersistentVars.rates[1] := 3300;
PersistentVars.rates[2] := 2300;
PersistentVars.rates[3] := 1500;
PersistentVars.rates[4] := 2400;
PersistentVars.rates[5] := 3600;
PersistentVars.rates[6] := 2700;
PersistentVars.rates[7] := 100;
*)

dwCRC := CRC32Finish(ulCRC:= CRC32Update(ulCRC:= CRC32Init(), pData:= pRetainArea, ulSize:= RetainAreaSize));

IF ((dwCRC <> dwCRCSave) OR R_TRIG1.Q) THEN
   IF NOT TOF1.Q OR R_TRIG1.Q THEN
      RTSIECResult := AppStoreRetainsInFile(pCurrentApp, pRetainFilePathName^); // записать в файл
		msg := "Save Ratains in file";
		PLC_PRG.logger.debug(msg);
	  
      IF RTSIECResult = 0 THEN
		msg := "Ratains saved Ok";
		PLC_PRG.logger.debug(msg);
         dwCRCSave := dwCRC;         
		 SysProcessExecuteCommand(synccmd, ADR(RTSIECResult) );
		msg := "Sync Ratains ret=";
		msg := WCONCAT(msg, UDINT_TO_WSTRING(RTSIECResult));
		PLC_PRG.logger.debug(msg);
	   ELSE
		msg := "Ratains saved Error=";
		msg := WCONCAT(msg, UDINT_TO_WSTRING(RTSIECResult));
		PLC_PRG.logger.debug(msg);
      END_IF
      AttemptSaveCounter := AttemptSaveCounter + 1;
		msg := "Retains: AttemptSaveCounter=";
		msg := WCONCAT(msg, INT_TO_WSTRING(AttemptSaveCounter));
		PLC_PRG.logger.debug(msg);
      TOF1(IN := TRUE);
   END_IF
END_IF

IF TOF1.Q THEN
   TOF1(IN := FALSE);
END_IF

END_PROGRAM

// CompWin/AppTerminalPost/Post/Post
// Моечный пост
FUNCTION_BLOCK PUBLIC Post
VAR_INPUT
//	InBanknote:	REAL;
//	InCoin:	REAL;
END_VAR
VAR_OUTPUT
	sVersion: 					STRING;	//ВерсияПО ()
	uIDTerminal:				UINT;	//Адрес терминала ()

	rAmountFreeWash:			REAL;	//Однократная сумма бесплатной мойки (руб)

	bCleeningPost: 				BOOL;	//Признак уборки (флаг)
	rEnteredCashAmount: 		REAL;	//Внесенная сумма (руб)
	rAmountOfCheck: 			REAL;	//Сумма для чека (руб)
	eStateTerminal: 			EnumStatePost;	//Состояние Терминала ()
	timRemainingTimeMode1: 		TIME;	//Оставшиеся время режима Р1 (c)
	timRemainingTimeMode2: 		TIME;	//Оставшиеся время режима Р2 (c)
	timRemainingTimeMode3: 		TIME;	//Оставшиеся время режима Р3 (c)
	timRemainingTimeMode4: 		TIME;	//Оставшиеся время режима Р4 (c)
	timRemainingTimeMode5: 		TIME;	//Оставшиеся время режима Р5 (c)
	timRemainingTimeMode6: 		TIME;	//Оставшиеся время режима Р6 (c)
	timRemainingTimeMode7: 		TIME;	//Оставшиеся время режима Р7 (c)
	timRemainingTimePause: 		TIME;	//Оставшиеся время режима Пауза (c)
	uCountBankNote: 			UINT;	//Счётчик купюр в ChashBox (шт)
	uCountCoin: 				UINT;	//Счётчик монет в ChashBox (шт)
	uNumberNotTransferredData: 	UINT;	//Количество не преданнных данных (пакет)

//	eCommandWashingMode: 		EnumMode;	//Сигнал включения функции мойки   ()	
	Mode: 		EnumMode := EnumMode.IDLE;	//Сигнал включения функции мойки   ()
	ModeStartTime : DT;	
	
	// стоимость мойки
	costWash: REAL := 0;
	
	// журнал стоимости текущей (прошлой) мойки
	ModesLog: ARRAY [1 .. 14] OF EventMode;

//	ModesLog: ARRAY [EnumMode.ACTIVECLEAN .. EnumMode.PAUSE] OF EventMode;
	ModePaid: BOOL := TRUE;	// Признак платной мойки
	
	ModeFinInfo: STRING(255);
	FinCostSummary: STRING;
	FinCostChange: STRING;
	
	InCash: REAL;
	InCard: REAL;
	CounterFund: REAL;
	Received: WORD;
	lastInCash : REAL;
END_VAR

VAR
	Number:						INT;	// номер поста
	messageCard :WSTRING;
	
	// Карта
	ActiveCardType: EnumCardType := EnumCardType.UNDEFINED;	
	ActiveCard : STRING[8] := ''; // cardId первые 4 байта

	// Состояние замков
	Locks : ARRAY [EnumLock.LOCK_TOP .. EnumLock.LOCK_MID] OF BOOL := [2(TRUE)];
	
	messageCollectcash1 :WSTRING;
	messageCollectcash2 :WSTRING;
	messageCollectcash3 :WSTRING;
	
	// Добавление бесплатных денег
	messageFreemoney1 :WSTRING;
	messageFreemoney2 :WSTRING;
	messageFreemoney3 :WSTRING;
	messageFreemoney4 :WSTRING;	
	messageFreemoney5 :WSTRING;	
	
	// текущий процент бонуса
	currentBonus: WORD := 0;
END_VAR

StartWash();

METHOD PUBLIC ChangeMode : EnumMode
VAR_INPUT
	newMode : EnumMode;
END_VAR
VAR
	durationMs: TIME;
	durationSecond: DWORD;
	message: STRING[512];
END_VAR
IF(Mode <> newMode)THEN
	// перед началом новой мойки сбросить журнал прошлой мойки
	IF(newMode = EnumMode.FUNC)THEN
		StartWash();
	END_IF
	
	IF((Mode >= EnumMode.ACTIVECLEAN AND Mode <= EnumMode.PAUSE) OR (Mode = EnumMode.HIGHPRESSURE))THEN
		// запомнить время окончания режима
		ModesLog[Mode].StopMode(inStopTime := PLC_PRG.GetCurrentTime(), rate := GetRates(Mode));

		// запомнить строку прошедшего режима, но не для сервисного режима
		IF(PLC_PRG.post.ActiveCardType <> EnumCardType.SERVICE)THEN
			// запомнить строку прошедшей функции
			//PersistentVars.messageFunc := "funcId=1; func=ACTIVECLEAN; cost=1234.56; paid=0; dur=3600; cardID=ABCDEF10; cardType=1; bonus=30;"
			// 8; PAUSE; 11.133334;
	//		message := WORD_TO_WSTRING(Mode);
	//		message := WCONCAT(message, '; ');
			CASE Mode OF
				EnumMode.ACTIVECLEAN:
					message := CONCAT(message, 'funcId=1; func=ACTIVECLEAN; ');
				EnumMode.SHAMPOO:
					// подмена шампунь - пена
					message := CONCAT(message, 'funcId=3; func=FOAM; ');
				EnumMode.FOAM:
					// подмена шампунь - пена
					message := CONCAT(message, 'funcId=2; func=SHAMPOO; ');
				EnumMode.COLDWATER:
					message := CONCAT(message, 'funcId=4; func=COLDWATER; ');
				EnumMode.HOTWATER:
					message := CONCAT(message, 'funcId=5; func=HOTWATER; ');
				EnumMode.WAX:
					message := CONCAT(message, 'funcId=6; func=WAX; ');
				EnumMode.OSMOSE:
					message := CONCAT(message, 'funcId=7; func=OSMOSE; ');
				EnumMode.PAUSE:
					message := CONCAT(message, 'funcId=8; func=PAUSE; ');
				EnumMode.HIGHPRESSURE:
					message := CONCAT(message, 'funcId=14; func=HIGHPRESSURE; ');
			END_CASE
	
			// стоимость
			message := CONCAT(message, ' cost=');
	//		message := CONCAT(message, REAL_TO_STRING(ModesLog[Mode].Cost));
			message := CONCAT(message, OSCAT_BASIC.REAL_TO_STRF(ModesLog[Mode].Cost, 2, '.'));
			message := CONCAT(message, ';');
			
			// признак платности
			IF(ModesLog[Mode].Paid)THEN
				message := CONCAT(message, ' paid=1;');
			ELSE
				message := CONCAT(message, ' paid=0;');
			END_IF
	
			// продолжительность
			durationMs := ModesLog[Mode].StopTime - ModesLog[Mode].StartTime;
			durationSecond := TIME_TO_DWORD(durationMs / 1000);
	//		OSCAT_BASIC.DT_TO_STRF(durationSecond, 
			message := CONCAT(message, ' dur=');
			message := CONCAT(message, DWORD_TO_STRING(durationSecond));
			message := CONCAT(message, ';');
	
			// cardID
			message := CONCAT(message, ' cardID=');
			message := CONCAT(message, PLC_PRG.post.ActiveCard);
			message := CONCAT(message, ';');
			
			// cardType
			message := CONCAT(message, ' cardType=');
			message := CONCAT(message, WORD_TO_STRING(PLC_PRG.post.ActiveCardType));
			message := CONCAT(message, ';');
			
			// bonus
			message := CONCAT(message, ' bonus=');
			message := CONCAT(message, WORD_TO_STRING(PLC_PRG.post.currentBonus));
			message := CONCAT(message, ';');
			
			PersistentVars.messageFunc := message;
		END_IF
	END_IF

	Mode := newMode;
	ModeStartTime := PLC_PRG.currentTime;
	
	IF((Mode >= EnumMode.ACTIVECLEAN AND Mode <= EnumMode.PAUSE) OR (Mode = EnumMode.HIGHPRESSURE))THEN
		// запомнить время начала режима
		ModesLog[Mode].StartMode(inStartTime := PLC_PRG.GetCurrentTime(), inPaid := ModePaid);
		
//		// включить лампу нового режима
//		DeviceLamps.SetLamps(Mode, TRUE);
	
//		// включить лампу нового режима
//		IF(CounterFund > 0 OR NOT ModePaid)THEN
//			DeviceLamps.SetLamps(Mode, TRUE);
//		END_IF
	END_IF

	IF(newMode = EnumMode.FIN)THEN
		StopWash();
	END_IF
	
	IF(newMode = EnumMode.CASHCOLLECT)THEN
		BegCollectCash();
	END_IF
	
	IF(newMode = EnumMode.FREEMONEY)THEN
		BegFreemoney();
	END_IF
END_IF

DBG_PRG.SetMode(Mode);
END_METHOD

METHOD AddMoney : REAL
VAR_INPUT
	InBanknote: WORD;
	InCoin: WORD;
END_VAR
VAR
	message: STRING[512];
END_VAR
Received := InBanknote + InCoin;

InCash := InCash + Received;

// применить текущий бонус
CounterFund := CounterFund + Received + Received * (currentBonus / 100.0);

AddMoney := CounterFund;

IF(Received > 0)THEN
	//PersistentVars.CashFund := PersistentVars.CashFund + Received;
	PersistentVars.TotalFund := PersistentVars.TotalFund + Received;
	
	(*
	PersistentVars.totalBanknote10 := PersistentVars.totalBanknote10 + 
	PersistentVars.totalBanknote50 := PersistentVars.totalBanknote50 + 
	PersistentVars.totalBanknote100 := PersistentVars.totalBanknote100 + 
	PersistentVars.totalBanknote500 := PersistentVars.totalBanknote500 + 
	PersistentVars.totalBanknote1k := PersistentVars.totalBanknote1k + 

	PersistentVars.totalCoin10 := PersistentVars.totalCoin10 + 
	*)
	
	//PersistentVars.messageTotal := "total; b10=12345678; b50=12345678; b100=12345678; b500=12345678; b1K=12345678; m10=12345678;"
	message := 'total; ';

	message := CONCAT(message, 'b10=');
	message := CONCAT(message, DWORD_TO_STRING(PersistentVars.totalBanknote10));
	message := CONCAT(message, '; ');
	
	message := CONCAT(message, 'b50=');
	message := CONCAT(message, DWORD_TO_STRING(PersistentVars.totalBanknote50));
	message := CONCAT(message, '; ');
	
	message := CONCAT(message, 'b100=');
	message := CONCAT(message, DWORD_TO_STRING(PersistentVars.totalBanknote100));
	message := CONCAT(message, '; ');
	
	message := CONCAT(message, 'b500=');
	message := CONCAT(message, DWORD_TO_STRING(PersistentVars.totalBanknote500));
	message := CONCAT(message, '; ');
	
	message := CONCAT(message, 'b1K=');
	message := CONCAT(message, DWORD_TO_STRING(PersistentVars.totalBanknote1k));
	message := CONCAT(message, '; ');
	
	message := CONCAT(message, 'm10=');
	message := CONCAT(message, DWORD_TO_STRING(PersistentVars.totalCoin10));
	message := CONCAT(message, ';');
	
	PersistentVars.messageTotal := message;


	
	//PersistentVars.messageInCash := "InCash=%d; s=0; Banknote: b10=1; b50=2; b100=3; b500=4; b1K=5; b5K=6; Coin: m1=7; m2=8; m5=9; m10=10;"
	message := 'InCash=';
	message := CONCAT(message, WORD_TO_STRING(Received));
	message := CONCAT(message, ';');
	
	message := CONCAT(message, 's=');
	message := CONCAT(message, WORD_TO_STRING(GeFundFromCollect()));
	message := CONCAT(message, '; ');
	
	message := CONCAT(message, ' Banknote: ');
	message := CONCAT(message, 'b10=');
	message := CONCAT(message, WORD_TO_STRING(DeviceBanknote.GetCounterBanknote(10)));
	message := CONCAT(message, '; ');
	
	message := CONCAT(message, 'b50=');
	message := CONCAT(message, WORD_TO_STRING(DeviceBanknote.GetCounterBanknote(50)));
	message := CONCAT(message, '; ');
	
	message := CONCAT(message, 'b100=');
	message := CONCAT(message, WORD_TO_STRING(DeviceBanknote.GetCounterBanknote(100)));
	message := CONCAT(message, '; ');
	
	message := CONCAT(message, 'b500=');
	message := CONCAT(message, WORD_TO_STRING(DeviceBanknote.GetCounterBanknote(500)));
	message := CONCAT(message, '; ');
	
	message := CONCAT(message, 'b1K=');
	message := CONCAT(message, WORD_TO_STRING(DeviceBanknote.GetCounterBanknote(1000)));
	message := CONCAT(message, '; ');
	
	message := CONCAT(message, 'b5K=');
	message := CONCAT(message, WORD_TO_STRING(DeviceBanknote.GetCounterBanknote(5000)));
	message := CONCAT(message, ';');
	
	message := CONCAT(message, ' Coin: ');
	message := CONCAT(message, 'm1=');
	message := CONCAT(message, WORD_TO_STRING(DeviceCoin.GetCounterCoin(1)));
	message := CONCAT(message, '; ');
	
	message := CONCAT(message, 'm2=');
	message := CONCAT(message, WORD_TO_STRING(DeviceCoin.GetCounterCoin(2)));
	message := CONCAT(message, '; ');
	
	message := CONCAT(message, 'm5=');
	message := CONCAT(message, WORD_TO_STRING(DeviceCoin.GetCounterCoin(5)));
	message := CONCAT(message, '; ');
	
	message := CONCAT(message, 'm10=');
	message := CONCAT(message, WORD_TO_STRING(DeviceCoin.GetCounterCoin(10)));
	message := CONCAT(message, ';');
	
	PersistentVars.messageInCash := message;
END_IF
END_METHOD

METHOD PUBLIC RemAmount : REAL
VAR_INPUT
	i_second : DWORD;
END_VAR
VAR
	amount : REAL;
	fund : REAL;
END_VAR
IF(CounterFund > 0 AND ((Mode >= EnumMode.ACTIVECLEAN AND Mode <= EnumMode.PAUSE) OR (Mode = EnumMode.HIGHPRESSURE)))THEN
	IF(DataFromSpk.GetAllowedMode(INT_TO_BYTE(Mode)))THEN
		// уменьшать баланс только если функция без аварии от СПК 
		
		// пересчитать тариф текущего режима за секунду
		amount := GetRates(Mode) / 60.0;
		// вычислить отработанные за i_second рубли 
		amount := DWORD_TO_REAL(i_second) * amount;	
	
		// уменьшить баланс
		fund := CounterFund - amount;
		IF(fund <= 0)THEN
			fund := 0;
			ChangeMode(EnumMode.FIN);
		END_IF
		
		// в CounterFund реальное значение, отображаться через формат %d будет округленное до ближайшего целого
		CounterFund := fund;
		//CounterFund := DINT_TO_WORD(TRUNC(fund));	// отбросить дробную часть
		//CounterFund := REAL_TO_WORD(fund);	// округление до ближайшего целого
	END_IF
	
	RemAmount := CounterFund;
END_IF
END_METHOD

METHOD PUBLIC ResetModes : BOOL
VAR_INPUT
END_VAR
VAR
	mode: BYTE;
END_VAR
FOR mode := 1 TO 14 DO
	ModesLog[mode].ResetValues();
END_FOR

ModeFinInfo := '';
END_METHOD

METHOD FormatModeFinInfo : STRING
VAR_INPUT
END_VAR
VAR
	imode: EnumMode;
	//workSecond: DWORD;
	//amount: REAL;
END_VAR
ModeFinInfo := '';
costWash := 0;

FOR imode := EnumMode.ACTIVECLEAN TO EnumMode.PAUSE DO
	//IF(ModesLog[imode].StopTime <> ModesLog[imode].StartTime)THEN
	IF(ModesLog[imode].Cost > 0)THEN
		costWash := costWash + ModesLog[imode].Cost;
		//workSecond := TIME_TO_DWORD(ModesLog[imode].StopTime - ModesLog[imode].StartTime) / 1000;
		//// пересчитать тариф текущего режима за секунду
		//amount := rates[imode] / 60;
		//// вычислить отработанные за i_second рубли 
		//amount := DWORD_TO_REAL(workSecond) * amount;	
		CASE imode OF
			EnumMode.ACTIVECLEAN:
				IF(ModeFinInfo <> '')THEN
					ModeFinInfo := CONCAT(ModeFinInfo, '$R');
				END_IF
				ModeFinInfo := CONCAT(ModeFinInfo, 'ECO-power $T');
				ModeFinInfo := CONCAT(ModeFinInfo, REAL_TO_STRING(ModesLog[imode].Cost));
			EnumMode.FOAM:
				IF(ModeFinInfo <> '')THEN
					ModeFinInfo := CONCAT(ModeFinInfo, '$R');
				END_IF
				ModeFinInfo := CONCAT(ModeFinInfo, 'Пена $T');
				ModeFinInfo := CONCAT(ModeFinInfo, REAL_TO_STRING(ModesLog[imode].Cost));
			EnumMode.SHAMPOO:
				IF(ModeFinInfo <> '')THEN
					ModeFinInfo := CONCAT(ModeFinInfo, '$R');
				END_IF
				ModeFinInfo := CONCAT(ModeFinInfo, 'Шампунь $T');
				ModeFinInfo := CONCAT(ModeFinInfo, REAL_TO_STRING(ModesLog[imode].Cost));
			EnumMode.COLDWATER:
				IF(ModeFinInfo <> '')THEN
					ModeFinInfo := CONCAT(ModeFinInfo, '$R');
				END_IF
				ModeFinInfo := CONCAT(ModeFinInfo, 'Холодная вода $T');
				ModeFinInfo := CONCAT(ModeFinInfo, REAL_TO_STRING(ModesLog[imode].Cost));
			EnumMode.HOTWATER:
				IF(ModeFinInfo <> '')THEN
					ModeFinInfo := CONCAT(ModeFinInfo, '$R');
				END_IF
				ModeFinInfo := CONCAT(ModeFinInfo, 'Горячая вода $T');
				ModeFinInfo := CONCAT(ModeFinInfo, REAL_TO_STRING(ModesLog[imode].Cost));
			EnumMode.WAX:
				IF(ModeFinInfo <> '')THEN
					ModeFinInfo := CONCAT(ModeFinInfo, '$R');
				END_IF
				ModeFinInfo := CONCAT(ModeFinInfo, 'Воск $T');
				ModeFinInfo := CONCAT(ModeFinInfo, REAL_TO_STRING(ModesLog[imode].Cost));
			EnumMode.OSMOSE:
				IF(ModeFinInfo <> '')THEN
					ModeFinInfo := CONCAT(ModeFinInfo, '$R');
				END_IF
				ModeFinInfo := CONCAT(ModeFinInfo, 'Осмос $T');
				ModeFinInfo := CONCAT(ModeFinInfo, REAL_TO_STRING(ModesLog[imode].Cost));
			EnumMode.PAUSE:
				IF(ModeFinInfo <> '')THEN
					ModeFinInfo := CONCAT(ModeFinInfo, '$R');
				END_IF
				ModeFinInfo := CONCAT(ModeFinInfo, 'Пауза $T');
				ModeFinInfo := CONCAT(ModeFinInfo, REAL_TO_STRING(ModesLog[imode].Cost));
		END_CASE
	END_IF
	//ModesLog[mode].inMode := mode;
	//ModesLog[mode].inStartTime := DT#1970-01-01-00:00;
	//ModesLog[mode].inStopTime := DT#1970-01-01-00:00;
	//ModesLog[mode].inPaid := FALSE;
END_FOR

// Общая стоимость мойки
FinCostSummary := 'Итого $T$T';
FinCostSummary := CONCAT(FinCostSummary, REAL_TO_STRING(costWash));

(*
// Сдача
IF(InCash > costWash)THEN
	FinCostChange := 'Оплачено ';
	FinCostChange := CONCAT(FinCostChange, REAL_TO_STRING(InCash));
	FinCostChange := CONCAT(FinCostChange, ' р,$R');
	FinCostChange := CONCAT(FinCostChange, 'сдача ');
	FinCostChange := CONCAT(FinCostChange, REAL_TO_STRING(InCash - costWash));
	FinCostChange := CONCAT(FinCostChange, ' р.');
//	FinCostChange := CONCAT(FinCostChange, ' р зачислена на карту.');
END_IF
*)

FormatModeFinInfo := ModeFinInfo;
END_METHOD

METHOD PUBLIC StartWash : BOOL
VAR_INPUT
END_VAR
// сбросить стоимость мойки
costWash := 0;

// сбросить стоимость последней мойки
PLC_PRG.post.SetLastInCash(0);

ResetModes();

ModeFinInfo := '';
FinCostSummary := '';
FinCostChange := '';

//InCash := 0;
//InCard := 0;
//CounterFund := 0;
//Received := 0;

// запомнить теущий бонус
IF(currentBonus = 0)THEN
	currentBonus := DataFromSpk.GetBonusValue();
	
	// применить бонусы к начальному балансу мойки. Сначала вызывается Post.AddMoney, а затем Post.StartWash
	// бонусы к последующим внесениям в процессе мойки применяются в Post.AddMoney
	CounterFund := CounterFund + CounterFund * (currentBonus / 100.0);	
END_IF
END_METHOD

METHOD PUBLIC StopWash : BOOL
VAR_INPUT
END_VAR
VAR
	imode: EnumMode;	

	i: EnumButton;
END_VAR
CounterFund := 0;

IF(ModePaid)THEN
  // пересчитать стоимость мойки
  costWash := 0.0;
	FOR imode := 1 TO 14 DO
		IF(ModesLog[imode].Cost > 0)THEN
			costWash := costWash + ModesLog[imode].Cost;
		END_IF
	END_FOR
	
	ModeFinInfo := FormatModeFinInfo();
	
//	// печатать чек
//	IF(costWash > 0)THEN
//		SysTimeRtcConvertUtcToLocal(SysTimeRtcGet(udiResult), udiTimeLocal);
//		timeDate:= UDINT_TO_DT(udiTimeLocal);
//		DevicePrinter.PrintBill(printingTime := OSCAT_BASIC.UTC_TO_LTIME(timeDate, DST_ENABLE :=0, TIME_ZONE_OFFSET:=DevicePrinter.TIME_ZONE_MINUTES_OFFSET), costWash := costWash);
//	END_IF
ELSE
	// для уборки сразу перейти к экрану ожидания
	Mode := EnumMode.IDLE;
END_IF

ModePaid := TRUE;

// запомнить сумму последнего внесения
lastInCash := InCash;

// сбросить внесения для следующей мойки
InCash := 0;

// вернуть карту
DeviceCard.UnLockCard();

// Погасить кнопки
//FOR i := EnumButton.BTN_ACTIVECLEAN TO EnumButton.BTN_HELP DO
FOR i := 1 TO 10 DO
	DeviceLamps.SetLamps(i, FALSE);
END_FOR;

// сбросить теущий бонус
currentBonus := 0;
END_METHOD

METHOD PUBLIC SetCard : BOOL
VAR_INPUT
	cType: EnumCardType;
	cardId : ARRAY [0..9] OF BYTE; // cardId первые 4 байта
END_VAR
SetCard := FALSE;
ActiveCardType := cType;
IF(cType <> EnumCardType.UNDEFINED)THEN
	ActiveCard := OSCAT_BASIC.BYTE_TO_STRH(cardId[0]);
	ActiveCard := CONCAT(ActiveCard, OSCAT_BASIC.BYTE_TO_STRH(cardId[1]));
	ActiveCard := CONCAT(ActiveCard, OSCAT_BASIC.BYTE_TO_STRH(cardId[2]));
	ActiveCard := CONCAT(ActiveCard, OSCAT_BASIC.BYTE_TO_STRH(cardId[3]));
ELSE
	ActiveCard := '';
END_IF

IF(cType = EnumCardType.UNDEFINED)THEN
	// если карта пропала во время уборки, то закончить уборку
	IF(NOT ModePaid)THEN
		PLC_PRG.post.ChangeMode(EnumMode.IDLE);
		StopWash();
		ModePaid := TRUE;
	END_IF

	//SetCard := TRUE;
ELSIF(AvialableCardWork())THEN
	CASE cType OF
		// Уборка
		EnumCardType.CLEANUP:
			ModePaid := FALSE;
			//ChangeMode(EnumMode.FUNC);
			// Карта обработана
			SetCard := TRUE;

		// Инкассация
		EnumCardType.CASHCOLLECT:
			ChangeMode(EnumMode.CASHCOLLECT);
			// Карта обработана
			SetCard := TRUE;

		// Сервисная карта
		EnumCardType.SERVICE:
			ModePaid := FALSE;
			//ChangeMode(EnumMode.FUNC);
			// Карта обработана
			SetCard := TRUE;

//		// Карта добавления баланса
//		EnumCardType.FREEMONEY:
//			ChangeMode(EnumMode.FREEMONEY);
//			// Карта обработана
//			SetCard := TRUE;
	END_CASE
//ELSE
//	SetCard := FALSE;
END_IF
END_METHOD

METHOD PUBLIC AvialableCardWork : BOOL
VAR_INPUT
END_VAR
// с каратми работать только если терминал свободен
AvialableCardWork := InWaitModes();
END_METHOD

// признак поста в состоянии ожидания начала мойки
METHOD PUBLIC InWaitModes : BOOL
VAR_INPUT
END_VAR
// пост в ожидании и готов к началу мойки
// если он в ожидании
// в рекламе
// или в экране окончания мойки
// или в экране окончания инкассации
InWaitModes := (Mode = EnumMode.IDLE OR Mode = EnumMode.ADVERT OR Mode = EnumMode.FIN OR Mode = EnumMode.CASHCOLLECT_FIN);
END_METHOD

METHOD PUBLIC IsUnlocked : BOOL
VAR_INPUT
	lock : EnumLock;
END_VAR
//IsUnlocked := NOT Locks[lock];

//IsUnlocked := FALSE;

IF(lock = EnumLock.LOCK_TOP)THEN
	IsUnlocked := ((UBRAIN1.bDOut1 AND 2#0100_0000) <> 0);
ELSIF(lock = EnumLock.LOCK_MID)THEN
	IsUnlocked := ((UBRAIN1.bDOut1 AND 2#1000_0000) <> 0);
END_IF
END_METHOD

METHOD PUBLIC UnLock : BOOL
VAR_INPUT
	lock :EnumLock;
	On : BOOL;
END_VAR;
VAR
END_VAR
// открыть замок
IF(lock = EnumLock.LOCK_TOP)THEN
	DeviceOut.SetOut(6, On);
ELSIF(lock = EnumLock.LOCK_MID)THEN
	DeviceOut.SetOut(7, On);
END_IF

//// сбросить выход
//DeviceOut.SetOut(INT_TO_BYTE(lock), FALSE);

IF(On)THEN
	CASE lock OF
		EnumLock.LOCK_TOP:
			messageCollectcash1 := "ECO - инкассировать купюрник";
		EnumLock.LOCK_MID:
			messageCollectcash2 := "Пена - инкассировта монетник";
	END_CASE
ELSE	
	CASE lock OF
		EnumLock.LOCK_TOP:
			messageCollectcash1 := "ECO - открыть верхнюю дверь";
		EnumLock.LOCK_MID:
			messageCollectcash2 := "Пена - открыть среднюю дверь";
	END_CASE
END_IF

Locks[lock] := NOT On;

UnLock := TRUE;
END_METHOD

// признак готовности поста к мойке
METHOD PUBLIC IsReadyToWash : BOOL
VAR_INPUT
END_VAR
// пост может начинать мойку
// если положительный баланс
// или в состоянии бесплатной мойки (режим уборки)
IsReadyToWash := ((CounterFund > 0 OR NOT ModePaid) and Mode <> EnumMode.FREEMONEY);
END_METHOD

// Инициализация поста
METHOD PUBLIC Init : BOOL
VAR_INPUT
END_VAR
// восстановить retain переменные
RestoreRetainVars();

// номер поста
Number := PersistentVars.postNumber;
//Number := 1;

// закрыть замки
UnLock(EnumLock.LOCK_TOP, FALSE);
UnLock(EnumLock.LOCK_MID, FALSE);

// сбросить мойку
StopWash();

//// разблокировать карту
//DeviceCard.UnLockCard();
END_METHOD

METHOD EndCollectCash : BOOL
VAR
	message: STRING[512];
	collectSum : WORD;
END_VAR
// закрыть замки
UnLock(EnumLock.LOCK_TOP, FALSE);
UnLock(EnumLock.LOCK_MID, FALSE);
			
// вернуть карту
DeviceCard.UnLockCard();

messageCollectcash1 := "";
messageCollectcash2 := "";

messageCollectcash3 := "";

messageCard := "Заберите карту";

ChangeMode(EnumMode.CASHCOLLECT_FIN);

//PersistentVars.CashFund := 0;

//PersistentVars.messageInCash := "Collect s=0; Banknote: b10=1; b50=2; b100=3; b500=4; b1K=5; b5K=6; Coin: m1=7; m2=8; m5=9; m10=10;"
collectSum := 10*PersistentVars.counterBefCollectBanknote10 + 50*PersistentVars.counterBefCollectBanknote50 + 100*PersistentVars.counterBefCollectBanknote100 + 500*PersistentVars.counterBefCollectBanknote500 + 1000*PersistentVars.counterBefCollectBanknote1000;
collectSum := collectSum + 10*PersistentVars.counterBefCollectCoin10;
message := 'Collect; ';
message := CONCAT(message, 's=');
message := CONCAT(message, WORD_TO_STRING(collectSum));
message := CONCAT(message, '; ');

	message := CONCAT(message, ' Banknote: ');
	message := CONCAT(message, 'b10=');
	message := CONCAT(message, WORD_TO_STRING(PersistentVars.counterBefCollectBanknote10));
	message := CONCAT(message, '; ');
	
	message := CONCAT(message, 'b50=');
	message := CONCAT(message, WORD_TO_STRING(PersistentVars.counterBefCollectBanknote50));
	message := CONCAT(message, '; ');
	
	message := CONCAT(message, 'b100=');
	message := CONCAT(message, WORD_TO_STRING(PersistentVars.counterBefCollectBanknote100));
	message := CONCAT(message, '; ');
	
	message := CONCAT(message, 'b500=');
	message := CONCAT(message, WORD_TO_STRING(PersistentVars.counterBefCollectBanknote500));
	message := CONCAT(message, '; ');
	
	message := CONCAT(message, 'b1K=');
	message := CONCAT(message, WORD_TO_STRING(PersistentVars.counterBefCollectBanknote1000));
	message := CONCAT(message, '; ');
	
	message := CONCAT(message, ' Coin: ');
	message := CONCAT(message, 'm10=');
	message := CONCAT(message, WORD_TO_STRING(PersistentVars.counterBefCollectCoin10));
	message := CONCAT(message, ';');

PersistentVars.messageCollect := message;
END_METHOD

METHOD BegCollectCash : BOOL
VAR_INPUT
END_VAR
messageCollectcash1 := "ECO - открыть верхнюю дверь";
messageCollectcash2 := "Пена - открыть среднюю дверь";

messageCollectcash3 := "Пауза - вернуть карту";

messageCard := "";

//PersistentVars.messageCollectBanknote := 'Banknote: 10=0; 50=0; 100=0; 500=0; 1K=0; 5K=0;';
//PersistentVars.messageCollectCoin := 'Coin: 1=0; 2=0; 5=0; 10=0;';
	PersistentVars.counterBefCollectBanknote10 := 0;
	PersistentVars.counterBefCollectBanknote50 := 0;
	PersistentVars.counterBefCollectBanknote100 := 0;
	PersistentVars.counterBefCollectBanknote500 := 0;
	PersistentVars.counterBefCollectBanknote1000 := 0;

	PersistentVars.counterBefCollectCoin10 := 0;
END_METHOD

METHOD EndFreemoney : BOOL
VAR_INPUT
END_VAR
// вернуть карту
DeviceCard.UnLockCard();

messageFreemoney1 := "";
messageFreemoney2 := "";
messageFreemoney3 := "";
messageFreemoney4 := "";

messageFreemoney5 := "";

messageCard := "Заберите карту";

ChangeMode(EnumMode.IDLE);
END_METHOD

METHOD BegFreemoney : BOOL
VAR_INPUT
END_VAR
messageFreemoney1 := "ECO - добавить 5 рублей";
messageFreemoney2 := "Пена - добавить 10 рублей";
messageFreemoney3 := "Шампунь - добавить 50 рублей";
messageFreemoney4 := "Хол. вода - добавить 100 рублей";	

messageFreemoney5 := "Пауза - вернуть карту";

messageCard := "";
END_METHOD

// признак поста в состоянии останова или аварий всех функций
METHOD InStopMode : BOOL
VAR_INPUT
END_VAR
// пост в останове от панели
// или есть запрет всех функций от панели

InStopMode := (Mode = EnumMode.STOP OR NOT DataFromSpk.GetAllowedMode(0));
END_METHOD

// была нажата кнопка "Завершить"
METHOD OnFinButton : BOOL
VAR
END_VAR
IF(IsReadyToWash())THEN
// работа в режиме мойки
	IF(Mode = EnumMode.FIN)THEN
//		// печатать чек
//		IF(InCash > 0)THEN
//			SysTimeRtcConvertUtcToLocal(SysTimeRtcGet(udiResult), udiTimeLocal);
//			timeDate:= UDINT_TO_DT(udiTimeLocal);
//			DevicePrinter.PrintBill(printingTime := OSCAT_BASIC.UTC_TO_LTIME(timeDate, DST_ENABLE :=0, TIME_ZONE_OFFSET:=DevicePrinter.TIME_ZONE_MINUTES_OFFSET), costWash := InCash);
//		END_IF
	ELSE
		ChangeMode(EnumMode.FIN);
	END_IF
ELSIF(Mode = EnumMode.CASHCOLLECT)THEN
// работа в режиме инкассации
	// закончить инкассацию
	EndCollectCash();
ELSIF(Mode = EnumMode.FREEMONEY)THEN
// работа в режиме добавления денег (бесплатной мойки)
	EndFreemoney();
END_IF
END_METHOD

METHOD GeFundFromCollect : UINT
VAR_INPUT
END_VAR
//GetCashFund := PersistentVars.CashFund;
//GetCashFund := DeviceBanknote.GetCounterBanknote(0) + DeviceCoin.GetCounterCoin(0);
GeFundFromCollect := 10*PersistentVars.counterBanknote10 + 50*PersistentVars.counterBanknote50 + 100*PersistentVars.counterBanknote100 + 500*PersistentVars.counterBanknote500 + 1000*PersistentVars.counterBanknote1000 + 10*PersistentVars.counterCoin10;
END_METHOD

// реакция на пропадание электропитания
METHOD OnLowPower : BOOL
VAR_INPUT
END_VAR
// сохранить retain переменные
SaveRetainVars();
END_METHOD

// сохранить retain переменные
METHOD SaveRetainVars : BOOL
VAR_INPUT
END_VAR
RetainManager(ForceRestore := FALSE, ForceSave := TRUE, ForceBalance := TRUE);
END_METHOD

// восстановить retain переменные
METHOD RestoreRetainVars : BOOL
VAR_INPUT
END_VAR
// если было сохранение
END_METHOD

// выключить контроллер
METHOD Shutdown : BOOL
VAR_INPUT
END_VAR
// отключить аккумулятор
DeviceOut.SetOut(DeviceOut.OUT_RELAY_BIT, FALSE);
END_METHOD

METHOD GetMessageInCash : ARRAY[0..64] OF WORD
VAR
	message : STRING[130];
	buf : ARRAY[0..129] OF BYTE;
	maxb: UINT;

	res: ARRAY[0..64] OF WORD;
	maxw: UINT;

	i : UINT;
END_VAR
//GetMessageInCash := PersistentVars.messageInCash;

message := PersistentVars.messageInCash;
//message := 'qw';
maxb := INT_TO_UINT( MIN(len(message), 130) );
OSCAT_BASIC._STRING_TO_BUFFER(message, 0, ADR(buf), maxb);

maxw := (maxb / 2);
maxw := MIN(maxw, 64);

FOR i := 0 TO maxw DO
	res[i] := OSCAT_BASIC.WORD_OF_BYTE(buf[2*i], buf[2*i+1]); //OSCAT_BASIC.SWAP_BYTE(buf[i]);
END_FOR

GetMessageInCash := res;
END_METHOD

METHOD GetMessageFunc : ARRAY[0..64] OF WORD
VAR
	message : STRING[130];
	buf : ARRAY[0..129] OF BYTE;
	maxb: UINT;

	res: ARRAY[0..64] OF WORD;
	maxw: UINT;

	i : UINT;
END_VAR
//GetMessageFunc := PersistentVars.messageFunc;

message := PersistentVars.messageFunc;
//message := 'qw';
maxb := INT_TO_UINT( MIN(len(message), 130));
OSCAT_BASIC._STRING_TO_BUFFER(message, 0, ADR(buf), maxb);

maxw := (maxb / 2);
maxw := MIN(maxw, 64);

FOR i := 0 TO maxw DO
	res[i] := OSCAT_BASIC.WORD_OF_BYTE(buf[2*i], buf[2*i+1]); //OSCAT_BASIC.SWAP_BYTE(buf[i]);
END_FOR

GetMessageFunc := res;
END_METHOD

METHOD GetMessageCollect : ARRAY[0..64] OF WORD
VAR
	message : STRING[130];
	buf : ARRAY[0..129] OF BYTE;
	maxb: UINT;

	res: ARRAY[0..64] OF WORD;
	maxw: UINT;

	i : UINT;
END_VAR
//GetMessageCollect := PersistentVars.messageCollect;

message := PersistentVars.messageCollect;
//message := 'qw';
maxb := INT_TO_UINT( MIN(len(message), 130)) ;
OSCAT_BASIC._STRING_TO_BUFFER(message, 0, ADR(buf), maxb);

maxw := (maxb / 2);
maxw := MIN(maxw, 64);

FOR i := 0 TO maxw DO
	res[i] := OSCAT_BASIC.WORD_OF_BYTE(buf[2*i], buf[2*i+1]); //OSCAT_BASIC.SWAP_BYTE(buf[i]);
END_FOR

GetMessageCollect := res;
END_METHOD

METHOD GetFundTotal : UINT
VAR_INPUT
END_VAR
GetFundTotal := PersistentVars.TotalFund;
END_METHOD

METHOD GetRates : REAL
VAR_INPUT
	mode : 	EnumMode;
END_VAR
VAR
	i : INT;
END_VAR
//GetRates := rates[Mode];

GetRates := 0;

CASE mode OF
	EnumMode.ACTIVECLEAN:
		GetRates := PersistentVars.rates[0] / 100.0;
	EnumMode.FOAM:
		GetRates := PersistentVars.rates[1] / 100.0;
	EnumMode.SHAMPOO:
		GetRates := PersistentVars.rates[2] / 100.0;
	EnumMode.COLDWATER:
		GetRates := PersistentVars.rates[3] / 100.0;
	EnumMode.HOTWATER:
		GetRates := PersistentVars.rates[4] / 100.0;
	EnumMode.WAX:
		GetRates := PersistentVars.rates[5] / 100.0;
	EnumMode.OSMOSE:
		GetRates := PersistentVars.rates[6] / 100.0;
	EnumMode.PAUSE:
		GetRates := PersistentVars.rates[7] / 100.0;
	EnumMode.HIGHPRESSURE:
		GetRates := PersistentVars.rates[8] / 100.0;
END_CASE

//// переделка под пену и шампунь
//IF(mode = EnumMode.FOAM)THEN
//	mode := EnumMode.SHAMPOO;
//ELSIF(mode = EnumMode.SHAMPOO)THEN
//	mode := EnumMode.FOAM;
//END_IF

//IF(mode >= EnumMode.ACTIVECLEAN AND mode <= EnumMode.PAUSE)THEN
//	i := WORD_TO_INT(mode) - 1;
//	GetRates := PersistentVars.rates[i] / 100.0;
//END_IF
END_METHOD

METHOD SaveNewRates : BOOL
PersistentVars.rates[0] := SPK_DATA.gi_rates[0];
PersistentVars.rates[1] := SPK_DATA.gi_rates[1];
PersistentVars.rates[2] := SPK_DATA.gi_rates[2];
PersistentVars.rates[3] := SPK_DATA.gi_rates[3];
PersistentVars.rates[4] := SPK_DATA.gi_rates[4];
PersistentVars.rates[5] := SPK_DATA.gi_rates[5];
PersistentVars.rates[6] := SPK_DATA.gi_rates[6];
PersistentVars.rates[7] := SPK_DATA.gi_rates[7];
PersistentVars.rates[8] := SPK_DATA.gi_rates[8];

SaveNewRates := TRUE;
END_METHOD

// признак нахождения поста в режиме платной мойки
METHOD InPaidWashMode : BOOL
InPaidWashMode := ((CounterFund > 0) and Mode <> EnumMode.FREEMONEY);
END_METHOD

// признак нахождения поста в режиме уборки
METHOD InClearWashMode : BOOL
InClearWashMode := ((NOT ModePaid) and ActiveCardType = EnumCardType.CLEANUP);
END_METHOD

METHOD GetMessageTotal : ARRAY[0..64] OF WORD
VAR
	message : STRING[130];
	buf : ARRAY[0..129] OF BYTE;
	maxb: INT;

	res: ARRAY[0..64] OF WORD;
	maxw: INT;

	i : INT;
END_VAR
//GetMessageTotal := PersistentVars.messageTotal;

message := PersistentVars.messageTotal;

maxb := MIN(len(message), 130);
OSCAT_BASIC._STRING_TO_BUFFER(message, 0, ADR(buf), INT_TO_UINT( maxb) );

maxw := (maxb / 2);
maxw := MIN(maxw, 64);

FOR i := 0 TO maxw DO
	res[i] := OSCAT_BASIC.WORD_OF_BYTE(buf[2*i], buf[2*i+1]);
END_FOR

GetMessageTotal := res;
END_METHOD

// признак нахождения поста в режиме сервиса
METHOD InServiceMode : BOOL
InServiceMode := (ActiveCardType = EnumCardType.SERVICE);
END_METHOD

METHOD SetSavedFund : BOOL
VAR_INPUT
	savedDT : DATE_AND_TIME;
	savedFund : real;
END_VAR
VAR
	ct : DATE_AND_TIME;
END_VAR
// проверить необходимость применения сохранённого баланса
ct := PLC_PRG.GetCurrentTime();
//IF((ct - savedDT) <= T#1H)THEN
	CounterFund := savedFund;
//END_IF
END_METHOD

METHOD SaveNewPause : BOOL
PersistentVars.pauseActiveClean := WORD_TO_TIME(1000 * SPK_DATA.gi_pauseActiveClean);
PersistentVars.pauseFoam := WORD_TO_TIME(1000 * SPK_DATA.gi_pauseFoam);
PersistentVars.pauseShampoo := WORD_TO_TIME(1000 * SPK_DATA.gi_pauseShampoo);

SaveNewPause := TRUE;
END_METHOD

METHOD GetPauseActiveClean : TIME
GetPauseActiveClean := PersistentVars.pauseActiveClean;
END_METHOD

METHOD GetPauseFoam : TIME
GetPauseFoam := PersistentVars.pauseFoam;
END_METHOD

METHOD GetPauseShampoo : TIME
GetPauseShampoo := PersistentVars.pauseShampoo;
END_METHOD

METHOD SetLastInCash
VAR_INPUT
	val: real;
END_VAR
lastInCash := val;
END_METHOD

END_FUNCTION_BLOCK

// CompWin/AppTerminalPost/Post/EventMode
// Запись о включении функции
FUNCTION_BLOCK PUBLIC EventMode
VAR_INPUT
	inMode: EnumMode;	// функции
	inStartTime: DT;	// время начало функции
	inStopTime: DT;	// время окончания функции
	inPaid: BOOL;		// признак платной мойки
END_VAR
VAR_OUTPUT
END_VAR
VAR
	Mode: EnumMode;	// функции
	StartTime: DT;	// время начало функции
	StopTime: DT;	// время окончания функции
	Paid: BOOL;		// признак платной мойки
	Cost:	REAL;	// стоимость функции
END_VAR

METHOD PUBLIC SetValues : BOOL
VAR_INPUT
	inMode: EnumMode;	// функции
	inStartTime: DT;	// время начало функции
	inStopTime: DT;	// время окончания функции
	inPaid: BOOL;		// признак платной мойки
	inCost: REAL;
END_VAR
Mode :=	inMode;
StartTime := inStartTime;
StopTime := inStopTime;
Paid := inPaid;
Cost := inCost;
END_METHOD

METHOD PUBLIC ResetValues : BOOL
VAR_INPUT
END_VAR
Mode := mode;
StartTime := DT#1970-01-01-00:00;
StopTime := DT#1970-01-01-00:00;
Paid := FALSE;
Cost := 0;
END_METHOD

METHOD PUBLIC StartMode : BOOL
VAR_INPUT
	inStartTime: DT;
	inPaid: BOOL;
END_VAR
StartTime := inStartTime;
Paid := inPaid;
END_METHOD

METHOD PUBLIC StopMode : BOOL
VAR_INPUT
	inStopTime: DT;
	rate: REAL;
END_VAR
VAR
	workSecond: DWORD;
	amount: REAL;	
END_VAR
StopTime := inStopTime;

// Запомнить стоимость функции
workSecond := TIME_TO_DWORD(StopTime - StartTime) / 1000;
// пересчитать тариф текущего режима за секунду
amount := rate / 60;
// вычислить отработанные за i_second рубли 
amount := DWORD_TO_REAL(workSecond) * amount;

// прибавить стоимость
Cost := Cost + amount;
END_METHOD

END_FUNCTION_BLOCK

// CompWin/AppTerminalPost/DevLamps/DeviceLamps
PROGRAM DeviceLamps
VAR CONSTANT
	LMP_ACTIVECLEAN :BYTE := 1;	// Р1. ECO-power
	LMP_FOAM :BYTE	:= 2;	// Р2. Пена
	LMP_SHAMPOO :BYTE := 3;	// Р3. Шампунь
	LMP_COLDWATER :BYTE := 4;	// Р4. Холодная вода
	LMP_HOTWATER :BYTE := 5;	// Р5. Горячая вода
	LMP_WAX :BYTE := 6;	// Р6. Воск
	LMP_OSMOSE :BYTE := 7;	// Р7. Осмос
	LMP_PAUSE :BYTE := 8;	// Пауза
	LMP_PRINT :BYTE := 9;	// Печать чека
	LMP_HELP :BYTE := 10;	// Вызов оператора
	
	OUT_LOCK_TOP: BYTE := 11;	// замок верхней двери
	OUT_LOCK_MDL: BYTE := 12;	// замок средней двери

	COLOR_NONE : BYTE := 0;
	COLOR_BLUE : BYTE := 1;
	COLOR_GREEN : BYTE := 2;
	COLOR_RED : BYTE := 3;
	COLOR_MAGENTA : BYTE := 4;
	COLOR_YELLOW : BYTE := 5;
	COLOR_LIGHTBLUE : BYTE := 6;
	COLOR_WHITE : BYTE := 7;
	
	ILLUMINATION_COLOR_NONE : BYTE := 0;	// 2#0000_0000
	ILLUMINATION_COLOR_BLUE : BYTE := 2;	// 2#0000_0010
	ILLUMINATION_COLOR_GREEN : BYTE := 4;	// 2#0000_0100
	ILLUMINATION_COLOR_RED : BYTE := 8;		// 2#0000_1000
	ILLUMINATION_COLOR_MAGENTA : BYTE := 10;// 2#0000_1010
	ILLUMINATION_COLOR_YELLOW : BYTE := 12;// 2#0000_1100
	ILLUMINATION_COLOR_LIGHTBLUE : BYTE := 6;	// 2#0000_0110
	ILLUMINATION_COLOR_WHITE : BYTE := 14;// 2#0000_1110
	
END_VAR
VAR
	Lamps : ARRAY [1 .. 12] OF BOOL := [
		FALSE,	// ECO-power
		FALSE,	// Пена
		FALSE,	// шампунь
		FALSE,	// Холодная вода
		FALSE,	// Горячая вода
		FALSE,	// Воск
		FALSE,	// Осмос
		FALSE,	// Пауза
		FALSE,	// Печать чека
		FALSE,	// Вызов оператора
		FALSE,	// замок верхней двери
		FALSE	// замок средней двери
	];		
END_VAR


// 
//UBRAIN1.bDOut1 := 16#31;

METHOD PUBLIC SetLamps : INT
VAR_INPUT
	Index: INT;
	On: BOOL;
END_VAR
// для ХВ ВД другая функция
IF(Index = 10) THEN
	SetLightTurbo(On);
END_IF

Lamps[Index] := On;
(*
IF(On)THEN
	UBRAIN1.bColorButton[Index] := 2;
ELSE
	UBRAIN1.bColorButton[Index] := 3;
END_IF
*)	
SetLamps := Index;

//IF(Index >= EnumButton.BTN_ACTIVECLEAN AND Index <= EnumButton.BTN_PAUSE)THEN
IF(Index >= 1 AND Index <= 8)THEN
	IF On THEN 
		IF(Index = EnumButton.BTN_PAUSE)THEN
			UBRAIN1.bColorButton[Index - 1] := COLOR_MAGENTA;
		ELSE
			UBRAIN1.bColorButton[Index - 1] := COLOR_GREEN;		
		END_IF
	ELSE
	// UBRAIN1.bColorButton[Index - 1] := COLOR_NONE;
	  UBRAIN1.bColorButton[Index - 1] := COLOR_WHITE;
	//  UBRAIN1.bColorButton[Index - 1] := COLOR_LIGHTBLUE;
	END_IF
END_IF
END_METHOD

METHOD PUBLIC SetAlarmLamps : INT
VAR_INPUT
	Index: INT;
END_VAR
VAR
	i :INT;
END_VAR
IF(Index >= 1 AND Index <= 8)THEN
	UBRAIN1.bColorButton[Index - 1] := COLOR_RED;
ELSE
	FOR i := 1 TO 8 DO
		UBRAIN1.bColorButton[i-1] := COLOR_RED;	
	END_FOR
END_IF
END_METHOD

// подсветка терминала
METHOD SetIllumination : BOOL
VAR_INPUT
	illuminationColor : BYTE;
END_VAR

VAR
	bDOut : byte;
END_VAR
//bDOut := UBRAIN1.bDOut1;
//
//// сбросить биты подсветк терминала
//bDOut := bDOut AND 2#1111_0001; 
//
//// установить заданный цвет
//bDOut := bDOut OR illuminationColor;

//UBRAIN1.bDOut1 := bDOut;
END_METHOD

METHOD SetLampColor : INT
VAR_INPUT
	Index: INT;
	color : BYTE;
END_VAR
SetLampColor := Index;

//IF(Index >= EnumButton.BTN_ACTIVECLEAN AND Index <= EnumButton.BTN_PAUSE)THEN
IF(Index >= 1 AND Index <= 8)THEN
	UBRAIN1.bColorButton[Index - 1] := color;
END_IF
END_METHOD

METHOD SetLightTurbo
VAR_INPUT
	bLightOn : BOOL;	
END_VAR
VAR
	bDOut : BYTE;
END_VAR
//bDOut := UBRAIN1.bDOut1;
IF bLightOn THEN
	UBRAIN1.bDOut1 := DWORD_TO_BYTE(PUTBIT(UBRAIN1.bDOut1, 1, TRUE));
ELSE
	UBRAIN1.bDOut1 := DWORD_TO_BYTE(PUTBIT(UBRAIN1.bDOut1, 1, FALSE));
END_IF
//UBRAIN1.bDOut1 := bDOut;
END_METHOD

END_PROGRAM

// CompWin/AppTerminalPost/Debug/DBG_PRG
PROGRAM DBG_PRG
VAR_INPUT
	dbgProcess: BOOL := FALSE;	// признак отладки	
END_VAR
VAR
	debugStruct: DebugStruct;
END_VAR


(*
// отладка
IF(DBG_PRG.dbgProcess)THEN
	// отладка купюрника
	IF(DBG_PRG.debugStruct.InBanknote > 0) THEN
		DeviceBanknote.DbgInBanknote();
	END_IF
	
	// отладка монетника
	IF(DBG_PRG.debugStruct.InCoin > 0) THEN
		DeviceCoin.DbgInCoin();
	END_IF
	
//	// отладка кнопок
//	DeviceButtons.DbgButton();

	// работать с картами только если это допустимо состоянием
//	IF(DBG_PRG.debugStruct.CardType <> EnumCardType.UNDEFINED)THEN
		DeviceCard.DbgSetCard();
//	END_IF
END_IF

*)

METHOD PUBLIC GetInCoin : WORD
GetInCoin := debugStruct.InCoin;

debugStruct.InCoin := 0;
END_METHOD

METHOD PUBLIC SetMode : EnumMode
VAR_INPUT
	newMode : EnumMode;
END_VAR
CASE newMode OF
	EnumMode.FUNC,
	EnumMode.ACTIVECLEAN,
	EnumMode.FOAM,
	EnumMode.SHAMPOO,
	EnumMode.COLDWATER,
	EnumMode.HOTWATER,
	EnumMode.WAX,
	EnumMode.OSMOSE,
	EnumMode.PAUSE:
//		VisuElems.CURRENTVISU := 'VisFunc';
	EnumMode.FIN:
//		VisuElems.CURRENTVISU := 'VisFin';
	EnumMode.IDLE:
//		VisuElems.CURRENTVISU := 'VisIdle';
	EnumMode.ADVERT:
//		VisuElems.CURRENTVISU := 'VisAdvert';
	EnumMode.CASHCOLLECT, EnumMode.CASHCOLLECT_FIN:
//		VisuElems.CURRENTVISU := 'VisCashCollect';		
	EnumMode.FREEMONEY:
//		VisuElems.CURRENTVISU := 'VisFreeMoney';
END_CASE

//debugStruct.Mode := newMode;
//SetMode := debugStruct.Mode;

SetMode := newMode;
END_METHOD

METHOD PUBLIC GetInBanknote : WORD
GetInBanknote := debugStruct.InBanknote;

debugStruct.InBanknote := 0;
END_METHOD

METHOD PUBLIC UnLockCard : BOOL
VAR_INPUT
END_VAR
DBG_PRG.debugStruct.CardType := EnumCardType.UNDEFINED;
END_METHOD

END_PROGRAM

// CompWin/AppTerminalPost/Cash/DeviceBanknote
PROGRAM DeviceBanknote
VAR
fb_COMcontrol: COM_CONTROL;
fb_CashCode: CashCode;
//fb_MV110_8A_DCON: MV110_8A_DCON;
//fb_SET_4TM : SET_4TM;
//i: INT;
xOpen: BOOL;
xClose: BOOL;

	amountReceived : WORD :=0;
	_amountReceivedTemp : WORD :=0;
	
	_isCollected: BOOL := FALSE;	// Признак проведённой инкассации для сброса количества купюр

	// состояние купюрника
	cashcodeStatus : WORD := 0;
	// ошибка купюрника
	cashcodeError : WORD := 0;

	// флаг снятия касетты
	casetteDropped : WORD := 0;
	// флаг зажёвывания банкноты
	banknoteJammed : WORD := 0;

	
	
	errCnt: UINT := 0;
	state : devBank := devBank.INIT;
	
END_VAR

CASE state OF
devBank.INIT: //init
	errCnt := 0;
	IF fb_COMcontrol.hCom > 0 THEN 
		state := devBank.CLOSE;
		ELSE
		state := devBank.OPEN;
			
	END_IF
 
devBank.CLOSE:
	xOpen:=FALSE;
	xClose := TRUE;
	fb_COMcontrol
	(
		xOpen := xOpen,
		xClose := xClose,
		uiPortNumber := 4,
		udiBaudrate := 9600,
		uiParity := COM.PARITY.NONE,
		uiByteSize := 8,
		uiStopBits := COM.STOPBIT.ONESTOPBIT
	);
	IF fb_COMcontrol.hCom = 0 THEN
		state := devBank.INIT;
	END_IF
devBank.OPEN: // открываем COM-порт COM2 (номер порта в CODESYS на +1 больше)
	xOpen:=TRUE;
	xClose := FALSE;
	
	fb_COMcontrol
	(
		xOpen := xOpen,
		xClose := xClose,
		uiPortNumber := 4,
		udiBaudrate := 9600,
		uiParity := COM.PARITY.NONE,
		uiByteSize := 8,
		uiStopBits := COM.STOPBIT.ONESTOPBIT
	);
	IF fb_COMcontrol.xDone AND fb_COMcontrol.hCom > 0 THEN
		state := devBank.PROCESS;
	END_IF
	
devBank.PROCESS: // опрашиваем модуль МВ110-8А по протоколу DCON
(* ???
IF(NOT (_isInitialized) AND PLC_PRG.comPortCascode > 0) THEN
// Инициализация купюрника
	//_device.init(iComPort := PLC_PRG.comPortCascode);
	_device.init(iComPort := PLC_PRG.comPortCascode, iBillTypes := BILL_10RUB OR BILL_50RUB OR BILL_100RUB );
	_isInitialized :=  TRUE;
END_IF;
*)
	fb_CashCode
	(
		xEnable := fb_COMcontrol.xDone,
		hCom := fb_COMcontrol.hCom,
		byAdress := 1
	);
	IF fb_CashCode.xDone THEN
		state := devBank.PROCESS;
		errCnt := 0;
	ELSE
		errCnt := errCnt + 1;
		IF errCnt > 1000 THEN 
			state := devBank.CLOSE;
		END_IF
	END_IF
//-----------------------------------------------	
	cashcodeStatus := fb_CashCode.Status.cashcodeStatus;
	cashcodeError := fb_CashCode.Status.cashcodeError;

	// считывание флага замятия
	banknoteJammed := fb_CashCode.Status.banknoteJammed;
	// считывание флага снятия кассеты
	casetteDropped := fb_CashCode.Status.casetteDropped;
//------------------------------------------------
(*
	IF (fb_CashCode.Status.error = CACHECODE_NO_ERROR AND NOT (fb_CashCode.Status.busy)) THEN
		// считывание флага замятия
		banknoteJammed := fb_CashCode.Status.banknoteJammed;
	
		// считывание флага снятия кассеты
		casetteDropped := fb_CashCode.Status.casetteDropped;
	END_IF
*)
(*
	IF (fb_CashCode.Status.error = CACHECODE_NO_ERROR AND NOT (fb_CashCode.Status.busy) AND fb_CashCode.Status.moneyReceived > 0) THEN
		// получить принятую сумму
		_amountReceivedTemp := _amountReceivedTemp + fb_CashCode.Status.moneyReceived;
		_amountReceivedTemp := fb_CashCode.Status.moneyReceived;
(*
		msg2 := "";
		msg2 := WCONCAT(msg2, "_amountReceivedTemp = ");
		msg2 := WCONCAT(msg2, WORD_TO_WSTRING(_amountReceivedTemp));
		msg2 := WCONCAT(msg2, "RUB");
		msg2 := WCONCAT(msg2, "   fb_CashCode.Status.moneyReceived = ");
		msg2 := WCONCAT(msg2, WORD_TO_WSTRING(fb_CashCode.Status.moneyReceived));
		msg2 := WCONCAT(msg2, "RUB");
		PLC_PRG.logger.debug(msg2);
*)		
		//countBanknote := countBanknote + _deviceStatus.countBanknote;
(*		
		PersistentVars.counterBanknote10 := PersistentVars.counterBanknote10 + fb_CashCode.Status.receivedBanknote10;
		PersistentVars.counterBanknote50 := PersistentVars.counterBanknote50 + fb_CashCode.Status.receivedBanknote50;
		PersistentVars.counterBanknote100 := PersistentVars.counterBanknote100 + fb_CashCode.Status.receivedBanknote100;
		PersistentVars.counterBanknote500 := PersistentVars.counterBanknote500 + fb_CashCode.Status.receivedBanknote500;
		PersistentVars.counterBanknote1000 := PersistentVars.counterBanknote1000 + fb_CashCode.Status.receivedBanknote1000;
		
		// увеличить тотальные счётчики номиналов
		PersistentVars.totalBanknote10 := PersistentVars.totalBanknote10 + fb_CashCode.Status.receivedBanknote10;
		PersistentVars.totalBanknote50 := PersistentVars.totalBanknote50 + fb_CashCode.Status.receivedBanknote50;
		PersistentVars.totalBanknote100 := PersistentVars.totalBanknote100 + fb_CashCode.Status.receivedBanknote100;
		PersistentVars.totalBanknote500 := PersistentVars.totalBanknote500 + fb_CashCode.Status.receivedBanknote500;
		PersistentVars.totalBanknote1k := PersistentVars.totalBanknote1k + fb_CashCode.Status.receivedBanknote1000;
		fb_CashCode.resetMoneyCnt();
*)
	END_IF
*)
(*
	// если внешней программой была обработана сумма, то перенести принятую сумму в прееменную для внешенй обработки
	IF(amountReceived = 0 AND _amountReceivedTemp > 0)THEN
		amountReceived := _amountReceivedTemp;
		_amountReceivedTemp := 0;
(*		
		msg3 := "";
		msg3 := WCONCAT(msg3, "amountReceived = ");
		msg3 := WCONCAT(msg3, WORD_TO_WSTRING(amountReceived));
		msg3 := WCONCAT(msg3, "RUB");
		msg3 := WCONCAT(msg3, "   _amountReceivedTemp = ");
		msg3 := WCONCAT(msg3, WORD_TO_WSTRING(_amountReceivedTemp));
		msg3 := WCONCAT(msg3, "RUB");
		PLC_PRG.logger.debug(msg3);
*)
	END_IF
*)
	// если внешней программой был сброшен счётчик купюр, то сбросить его внутри
	IF(_isCollected)THEN
		// запомнить значения счётчиков
		// только если было начало инкассации и счётчики ещё не сброшены
		// (защита от повторного нажатия кнопок инкассации)
		IF(PersistentVars.counterBefCollectBanknote10 = 0 AND PersistentVars.counterBefCollectBanknote50 = 0 AND PersistentVars.counterBefCollectBanknote100 = 0 AND PersistentVars.counterBefCollectBanknote500 = 0 AND PersistentVars.counterBefCollectBanknote1000 = 0) THEN
			PersistentVars.counterBefCollectBanknote10 := PersistentVars.counterBanknote10;
			PersistentVars.counterBefCollectBanknote50 := PersistentVars.counterBanknote50;
			PersistentVars.counterBefCollectBanknote100 := PersistentVars.counterBanknote100;
			PersistentVars.counterBefCollectBanknote500 := PersistentVars.counterBanknote500;
			PersistentVars.counterBefCollectBanknote1000 := PersistentVars.counterBanknote1000;
		END_IF

		// сбросить значения
		PersistentVars.counterBanknote10 := 0;
		PersistentVars.counterBanknote50 := 0;
		PersistentVars.counterBanknote100 := 0;
		PersistentVars.counterBanknote500 := 0;
		PersistentVars.counterBanknote1000 := 0;

		_isCollected := FALSE;
	END_IF
	
//-----------------------------------------------	
END_CASE

METHOD GetCounterBanknote : UINT
VAR_INPUT
	// номинал
	nom: INT;
END_VAR
GetCounterBanknote := 0;

CASE nom OF
	0:
		GetCounterBanknote := PersistentVars.counterBanknote10 + PersistentVars.counterBanknote50 + PersistentVars.counterBanknote100 + PersistentVars.counterBanknote500 + PersistentVars.counterBanknote1000;
	10:
		GetCounterBanknote := PersistentVars.counterBanknote10;
	50:
		GetCounterBanknote := PersistentVars.counterBanknote50;
	100:
		GetCounterBanknote := PersistentVars.counterBanknote100;
	500:
		GetCounterBanknote := PersistentVars.counterBanknote500;
	1000:
		GetCounterBanknote := PersistentVars.counterBanknote1000;
END_CASE
END_METHOD

METHOD IsCasetteDropped : WORD
IsCasetteDropped := casetteDropped;
END_METHOD

METHOD IsBanknoteJammed : WORD
VAR_INPUT
END_VAR
IsBanknoteJammed := banknoteJammed;
END_METHOD

// Инкассация устройства
METHOD PUBLIC CollectCash : UINT
VAR_INPUT
END_VAR
// выстаитьВыставить признка необходимости сброса счётчика купюр
_isCollected := TRUE;
END_METHOD

// Вернуть во вне принятую сумму, 
// затем сбросить сумму для записывания следующих принятий
METHOD PUBLIC GetReceived : WORD
VAR_INPUT
END_VAR
	
//GetReceived := amountReceived;
	IF fb_CashCode.Status.moneyReceived > 0 THEN 
		GetReceived := fb_CashCode.Status.moneyReceived;
		
		PersistentVars.counterBanknote10 := PersistentVars.counterBanknote10 + fb_CashCode.Status.receivedBanknote10;
		PersistentVars.counterBanknote50 := PersistentVars.counterBanknote50 + fb_CashCode.Status.receivedBanknote50;
		PersistentVars.counterBanknote100 := PersistentVars.counterBanknote100 + fb_CashCode.Status.receivedBanknote100;
		PersistentVars.counterBanknote500 := PersistentVars.counterBanknote500 + fb_CashCode.Status.receivedBanknote500;
		PersistentVars.counterBanknote1000 := PersistentVars.counterBanknote1000 + fb_CashCode.Status.receivedBanknote1000;
		
		// увеличить тотальные счётчики номиналов
		PersistentVars.totalBanknote10 := PersistentVars.totalBanknote10 + fb_CashCode.Status.receivedBanknote10;
		PersistentVars.totalBanknote50 := PersistentVars.totalBanknote50 + fb_CashCode.Status.receivedBanknote50;
		PersistentVars.totalBanknote100 := PersistentVars.totalBanknote100 + fb_CashCode.Status.receivedBanknote100;
		PersistentVars.totalBanknote500 := PersistentVars.totalBanknote500 + fb_CashCode.Status.receivedBanknote500;
		PersistentVars.totalBanknote1k := PersistentVars.totalBanknote1k + fb_CashCode.Status.receivedBanknote1000;
		
		fb_CashCode.resetMoneyCnt();
		fb_CashCode.resetMoneyReceived();
	END_IF


//amountReceived := 0;
END_METHOD

END_PROGRAM

// CompWin/AppTerminalPost/Cash/COM_CONTROL
FUNCTION_BLOCK COM_CONTROL
VAR_IN_OUT
xOpen: BOOL; // сигнал открытия порта
xClose: BOOL; // сигнал закрытия порта
END_VAR
VAR_INPUT
uiPortNumber: UINT; // номер порта
udiBaudrate: UDINT; // скорость передачи данных
uiParity: COM.PARITY; // четность
uiByteSize: UINT; // кол-во бит данных в байте
uiStopBits: COM.STOPBIT; // кол-во стоп бит
END_VAR
VAR_OUTPUT
xDone: BOOL; // флаг успешного открытия порта
hCom: COM.CAA.HANDLE; // дескриптор порта
xOpenError: BOOL; // флаг ошибки открытия порта
xCloseError: BOOL; // флаг ошибки закрытия порта
END_VAR
VAR
aComParams: ARRAY [1..5] OF COM.PARAMETER; // структура настроек порта
fb_COMopen: COM.Open; // ФБ открытия порта
fb_COMclose: COM.Close; // ФБ закрытия порта
eState: COM_STATE; // текущий шаг работы с портом
	
END_VAR


CASE eState OF
	INITIALIZE:
	10:
	
	
END_CASE


CASE eState OF
	INITIALIZE :
		fb_COMopen (xExecute:=FALSE);
		fb_COMclose (xExecute:=FALSE);
		eState:=WAITING_FOR_SIGNAL;
		
	WAITING_FOR_SIGNAL:
		IF xOpen THEN
			IF hCom=0 OR hCom=16#FFFFFFFF THEN
				eState := OPEN_PORT;
			ELSE
				xOpen := FALSE;
				xDone := TRUE;
				eState := INITIALIZE;
			END_IF
		END_IF
		IF xClose THEN
			IF hCom>0 AND hCom<16#FFFFFFFF THEN
				eState := CLOSE_PORT;
			ELSE
				xClose := FALSE;
				xDone := FALSE;
				eState := INITIALIZE;
			END_IF
		END_IF
	
	OPEN_PORT:
		SETTINGS();
		OPEN();
		IF fb_COMopen.xDone AND fb_COMopen.xExecute THEN
			xOpen := FALSE;
			fb_COMopen(xExecute:=FALSE);
			xDone := TRUE;
			eState := INITIALIZE;
		END_IF
		IF fb_COMopen.xError AND fb_COMopen.xExecute THEN
			xOpenError := TRUE;
			fb_COMopen(xExecute:=FALSE);
			xDone := FALSE;
			eState := INITIALIZE;
		END_IF

	CLOSE_PORT:
		CLOSE();
		IF fb_COMclose.xDone AND fb_COMclose.xExecute THEN
			xClose := FALSE;
			xDone := FALSE;
			hCom := 0;
			fb_COMclose(xExecute:=FALSE);
			eState := INITIALIZE;
		END_IF
			IF fb_COMclose.xError AND fb_COMclose.xExecute THEN
				xCloseError := TRUE;
				fb_COMclose(xExecute:=FALSE);
		END_IF
END_CASE

ACTION CLOSE:
fb_COMclose.hCom := hCom;
fb_COMclose.xExecute := TRUE;
fb_COMclose();
END_ACTION

ACTION OPEN:
fb_COMopen.usiListLength := UINT_TO_USINT(SIZEOF(aComParams) / SIZEOF(COM.PARAMETER));
fb_COMopen.pParameterList := ADR(aComParams);
fb_COMopen.xExecute := TRUE;
fb_COMopen();
hCom := fb_COMopen.hCom;
END_ACTION

ACTION SETTINGS:
aComParams[1].udiParameterId := COM.CAA_Parameter_Constants.udiPort;
aComParams[1].udiValue := uiPortNumber;
aComParams[2].udiParameterId := COM.CAA_Parameter_Constants.udiBaudrate;
aComParams[2].udiValue := udiBaudrate;
aComParams[3].udiParameterId := COM.CAA_Parameter_Constants.udiParity;
aComParams[3].udiValue := ANY_TO_UDINT(uiParity);
aComParams[4].udiParameterId := COM.CAA_Parameter_Constants.udiByteSize;
aComParams[4].udiValue := uiByteSize;
aComParams[5].udiParameterId := COM.CAA_Parameter_Constants.udiStopBits;
aComParams[5].udiValue := ANY_TO_UDINT(uiStopBits);
END_ACTION

END_FUNCTION_BLOCK

// CompWin/AppTerminalPost/Cash/CashCode
FUNCTION_BLOCK CashCode
VAR_INPUT
xEnable: BOOL; // сигнал опроса модуля
hCom: COM.CAA.HANDLE; // дескриптор COM-порта
byAdress: BYTE; // адрес опрашиваемого модуля
END_VAR
VAR_OUTPUT
	Status : cacheCodeStatus;	

xDone: BOOL; // флаг окончания текущего цикла опроса модуля
xWriteError: BOOL; // флаг ошибки отправки запроса
xReadError: BOOL; // флаг ошибки получения ответа
xTimeout: BOOL; // флаг отсутствия ответа по истечению таймаута опроса
xWrongCRC: BOOL; // флаг получения ответа с неправильной контрольной суммой


END_VAR
VAR
	eStateCCNET: CCNET_STATE := CCNET_STATE.INIT; // текущий шаг опроса модуля
	eStateCashCode: CASHCODE_STATE := CASHCODE_STATE.INIT; // текущий шаг опроса модуля
	fb_COMwrite: COM.Write; // ФБ отправки запроса
	fb_COMread: COM.Read; // ФБ получения ответа
//	sWriteData: STRING(255); // запрос к модулю в виде строки
//	sReadData: STRING(255); // полный ответ модуля в виде строки
//	sReadBuff: STRING(255); // часть ответа модуля

	sWriteData: ARRAY [0..255] OF BYTE; // запрос к модулю в виде строки
	sReadData: ARRAY [0..255] OF BYTE; // полный ответ модуля в виде строки
	sReadBuff: ARRAY [0..255] OF BYTE; // часть ответа модуля

	szWriteDataLen : COM.CAA.SIZE;;
	sAdress: STRING(2); // адрес опрашиваемого модуля в виде строки
	wCRC: WORD; // СRC
	sCRC: STRING(2); // СRC в виде строки
	xCorrectAnswer: BOOL; // флаг корректного (c верной CRC) ответа от модуля
	i: INT; // счетчик для цикла FOR
	fb_TON_Write: TON; // таймер
	fb_TON_Read: TON; // таймер
	fb_TON_Poll: TON;
	fb_ANALYZE_DATA: ANALYZE_DATA; // ФБ анализа ответа модуля
	szReadData : COM.CAA.SIZE;;
	szReadData1 : COM.CAA.SIZE;;
	szAnswerLen : COM.CAA.SIZE;;
	
	fl_disableCashCode: BOOL := FALSE;

	c_tTimeoutWrite: TIME:=T#40MS; // таймаут опроса модуля (время ожидания ответа)
	c_tTimeoutRead: TIME:=T#108MS; // таймаут опроса модуля (время ожидания ответа)
	c_tDelay: TIME:=T#200MS; // задержка перед отправкой следующего запроса
	Z1: BYTE := 0;
	Z2: BYTE := 0;
	cacheCodeConvertByteToMoney: UINT := 0;
	msg: WSTRING;
	sum: UINT := 0;
END_VAR

 

IF xEnable THEN
	
	

	CASE eStateCCNET OF
		CCNET_STATE.INIT:
			eStateCCNET := CCNET_STATE.IDLE;

		CCNET_STATE.IDLE:
			IF fl_disableCashCode THEN
				eStateCashCode := CASHCODE_STATE.DISABLE;
			END_IF

			CASE eStateCashCode OF
				CASHCODE_STATE.INIT:
					eStateCCNET := CCNET_STATE.SEND_RESET;
					
					eStateCashCode := CASHCODE_STATE.ENABLE_BILL_TYPES;
	
				CASHCODE_STATE.POLL:
					eStateCCNET := CCNET_STATE.SEND_POLL;

				CASHCODE_STATE.ENABLE_BILL_TYPES:
					eStateCCNET := CCNET_STATE.SEND_ENABLE_BILL_TYPES;
					eStateCashCode := CASHCODE_STATE.POLL;
	
